// TIA Portal V17 program export: 2 tag tables, 3 data types, 1 data blocks, 4 code blocks (in call order from the OBs), 2 instance data blocks

VAR_GLOBAL   // PLC tag table "Default tag table"
END_VAR

VAR_GLOBAL   // PLC tag table "LPMLV2022_Constants"
END_VAR
VAR_GLOBAL CONSTANT   // user constants
   LPMLV2022_MODE_INVALID : DInt := 0;   // OMAC PackMLV2022 unit mode Invalid
   LPMLV2022_MODE_PRODUCTION : DInt := 1;   // OMAC PackMLV2022 unit mode Production
   LPMLV2022_MODE_MAINTENANCE : DInt := 2;   // OMAC PackMLV2022 unit mode Maintenance
   LPMLV2022_MODE_MANUAL : DInt := 3;   // OMAC PackMLV2022 unit mode Manual
   LPMLV2022_MODE_USER_01 : DInt := 4;   // OMAC PackMLV2022 user-defined unit mode 01
   LPMLV2022_MODE_USER_02 : DInt := 5;   // OMAC PackMLV2022 user-defined unit mode 02
   LPMLV2022_MODE_USER_03 : DInt := 6;   // OMAC PackMLV2022 user-defined unit mode 03
   LPMLV2022_MODE_USER_04 : DInt := 7;   // OMAC PackMLV2022 user-defined unit mode 04
   LPMLV2022_MODE_USER_05 : DInt := 8;   // OMAC PackMLV2022 user-defined unit mode 05
   LPMLV2022_MODE_USER_06 : DInt := 9;   // OMAC PackMLV2022 user-defined unit mode 06
   LPMLV2022_MODE_USER_07 : DInt := 10;   // OMAC PackMLV2022 user-defined unit mode 07
   LPMLV2022_MODE_USER_08 : DInt := 11;   // OMAC PackMLV2022 user-defined unit mode 08
   LPMLV2022_MODE_USER_09 : DInt := 12;   // OMAC PackMLV2022 user-defined unit mode 09
   LPMLV2022_MODE_USER_10 : DInt := 13;   // OMAC PackMLV2022 user-defined unit mode 10
   LPMLV2022_MODE_USER_11 : DInt := 14;   // OMAC PackMLV2022 user-defined unit mode 11
   LPMLV2022_MODE_USER_12 : DInt := 15;   // OMAC PackMLV2022 user-defined unit mode 12
   LPMLV2022_MODE_USER_13 : DInt := 16;   // OMAC PackMLV2022 user-defined unit mode 13
   LPMLV2022_MODE_USER_14 : DInt := 17;   // OMAC PackMLV2022 user-defined unit mode 14
   LPMLV2022_MODE_USER_15 : DInt := 18;   // OMAC PackMLV2022 user-defined unit mode 15
   LPMLV2022_MODE_USER_16 : DInt := 19;   // OMAC PackMLV2022 user-defined unit mode 16
   LPMLV2022_MODE_USER_17 : DInt := 20;   // OMAC PackMLV2022 user-defined unit mode 17
   LPMLV2022_MODE_USER_18 : DInt := 21;   // OMAC PackMLV2022 user-defined unit mode 18
   LPMLV2022_MODE_USER_19 : DInt := 22;   // OMAC PackMLV2022 user-defined unit mode 19
   LPMLV2022_MODE_USER_20 : DInt := 23;   // OMAC PackMLV2022 user-defined unit mode 20
   LPMLV2022_MODE_USER_21 : DInt := 24;   // OMAC PackMLV2022 user-defined unit mode 21
   LPMLV2022_MODE_USER_22 : DInt := 25;   // OMAC PackMLV2022 user-defined unit mode 22
   LPMLV2022_MODE_USER_23 : DInt := 26;   // OMAC PackMLV2022 user-defined unit mode 23
   LPMLV2022_MODE_USER_24 : DInt := 27;   // OMAC PackMLV2022 user-defined unit mode 24
   LPMLV2022_MODE_USER_25 : DInt := 28;   // OMAC PackMLV2022 user-defined unit mode 25
   LPMLV2022_MODE_USER_26 : DInt := 29;   // OMAC PackMLV2022 user-defined unit mode 26
   LPMLV2022_MODE_USER_27 : DInt := 30;   // OMAC PackMLV2022 user-defined unit mode 27
   LPMLV2022_MODE_USER_28 : DInt := 31;   // OMAC PackMLV2022 user-defined unit mode 28
   LPMLV2022_STATE_UNDEFINED : DInt := 0;   // OMAC PackMLV2022 state Undefined
   LPMLV2022_STATE_CLEARING : DInt := 1;   // OMAC PackMLV2022 state Clearing
   LPMLV2022_STATE_STOPPED : DInt := 2;   // OMAC PackMLV2022 state Stopped
   LPMLV2022_STATE_STARTING : DInt := 3;   // OMAC PackMLV2022 state Starting
   LPMLV2022_STATE_IDLE : DInt := 4;   // OMAC PackMLV2022 state Idle
   LPMLV2022_STATE_SUSPENDED : DInt := 5;   // OMAC PackMLV2022 state Suspended
   LPMLV2022_STATE_EXECUTE : DInt := 6;   // OMAC PackMLV2022 state Execute
   LPMLV2022_STATE_STOPPING : DInt := 7;   // OMAC PackMLV2022 state Stopping
   LPMLV2022_STATE_ABORTING : DInt := 8;   // OMAC PackMLV2022 state Aborting
   LPMLV2022_STATE_ABORTED : DInt := 9;   // OMAC PackMLV2022 state Aborted
   LPMLV2022_STATE_HOLDING : DInt := 10;   // OMAC PackMLV2022 state Holding
   LPMLV2022_STATE_HELD : DInt := 11;   // OMAC PackMLV2022 state Held
   LPMLV2022_STATE_UNHOLDING : DInt := 12;   // OMAC PackMLV2022 state Unholding
   LPMLV2022_STATE_SUSPENDING : DInt := 13;   // OMAC PackMLV2022 state Suspending
   LPMLV2022_STATE_UNSUSPENDING : DInt := 14;   // OMAC PackMLV2022 state Unsuspending
   LPMLV2022_STATE_RESETTING : DInt := 15;   // OMAC PackMLV2022 state Resetting
   LPMLV2022_STATE_COMPLETING : DInt := 16;   // OMAC PackMLV2022 state Completing
   LPMLV2022_STATE_COMPLETED : DInt := 17;   // OMAC PackMLV2022 state Completed
   LPMLV2022_CMD_UNDEFINED : DInt := 0;   // OMAC PackMLV2022 control command Undefined
   LPMLV2022_CMD_RESET : DInt := 1;   // OMAC PackMLV2022 control command Reset
   LPMLV2022_CMD_START : DInt := 2;   // OMAC PackMLV2022 control command Start
   LPMLV2022_CMD_STOP : DInt := 3;   // OMAC PackMLV2022 control command Stop
   LPMLV2022_CMD_HOLD : DInt := 4;   // OMAC PackMLV2022 control command Hold
   LPMLV2022_CMD_UNHOLD : DInt := 5;   // OMAC PackMLV2022 control command Unhold
   LPMLV2022_CMD_SUSPEND : DInt := 6;   // OMAC PackMLV2022 control command Suspend
   LPMLV2022_CMD_UNSUSPEND : DInt := 7;   // OMAC PackMLV2022 control command Unsuspend
   LPMLV2022_CMD_ABORT : DInt := 8;   // OMAC PackMLV2022 control command Abort
   LPMLV2022_CMD_CLEAR : DInt := 9;   // OMAC PackMLV2022 control command Clear
   LPMLV2022_CMD_COMPLETE : DInt := 10;   // OMAC PackMLV2022 control command Complete
   LPMLV2022_DIAG_BUFFER_UPPER_LIM : Int := 7;   // Diagnostics buffer array upper boundary (0-based)
   LPMLV2022_MODES_UPPER_LIM : Int := 8;   // (Number of unit modes - 1) -> Array[0..LPMLV2022_MODES_UPPER_LIM]
   LPMLV2022_STATES_UPPER_LIM : Int := 17;   // (Number of states - 1) -> Array[0..LPMLV2022_STATES_UPPER_LIM]
   LPMLV2022_MAX_MODES_UPPER_LIM : Int := 31;   // (Maximum number of unit modes - 1) -> Array[0..LPMLV2022_MAX_MODES_UPPER_LIM]
END_VAR

TYPE "LPMLV2022_typeConfiguration"
TITLE = LPMLV2022_typeConfiguration
// Support: tech.team.motioncontrol@siemens.com
// stored: IsFailsafeCompliant false
   STRUCT
      EnabledModesCfg : DWord := 16#0000_01FE;   // Bit locations within the DWORD represent Mode numbers. A value of 1 in a bit location [0-31] indicates that the corresponding Mode number is enabled. Mode 0 is an Invalid Mode, therefore bit 0 is unused
      DisabledStatesCfg : Array[0.."LPMLV2022_MAX_MODES_UPPER_LIM"] of DWord;   // The array index represents the Mode number. Bit locations within the DWORD value represent State numbers. A value of 1 in a bit location indicates that the corresponding state number is disabled. State 0 is an Undefined State, therefore bit 0 is unused
      ModeTransitionCfg : Array[0.."LPMLV2022_MAX_MODES_UPPER_LIM"] of DWord;   // The array index represents the Mode number. Bit locations within the DWORD value represent State numbers. A value of 1 in a bit location indicates that a mode transition from the corresponding state number is allowed
      holdCmdCfg : DWord := 16#0000_0060;   // Bit locations within the DWORD value represent State numbers. A value of 1 in a bit location indicates that the Hold control command is taken into account in the corresponding state. Note: a state change is only performed if the Holding/Held states are not disabled. The 'holdCmdCfg' can only be activated for the following states: Idle, Starting, Execute, Completing, Completed, Suspending, Suspended, Unsuspending, Unholding
      completeCmdCfg : DWord := 16#0000_0860;   // Bit locations within the DWORD value represent State numbers. A value of 1 in a bit location indicates that the Complete control command is taken into account in the corresponding state. Note: a state change is only performed if the Completing/Completed states are not disabled. The 'completeCmdCfg' can only be activated for the following states: Execute, Suspended, Held
   END_STRUCT;
   // ModeTransitionCfg[1..31] := 16#0000_0214;
END_TYPE

TYPE "LPMLV2022_typeDiagnostics"
TITLE = LPMLV2022_typeDiagnostics
// Support: tech.team.motioncontrol@siemens.com
// stored: IsFailsafeCompliant false
   STRUCT
      bufferIndex { ExternalWritable := 'False'} : Int := -1;   // Index of actual buffer entry
      buffer { ExternalWritable := 'False'} : Array[0.."LPMLV2022_DIAG_BUFFER_UPPER_LIM"] of "LPMLV2022_typeDiagnosticsEntry";   // Diagnostics information buffer
   END_STRUCT;
END_TYPE

TYPE "LPMLV2022_typeDiagnosticsEntry"
TITLE = LPMLV2022_typeDiagnosticsEntry
// Support: tech.team.motioncontrol@siemens.com
// stored: IsFailsafeCompliant false
   STRUCT
      timestamp { ExternalWritable := 'False'} : DTL;   // Timestamp for this entry
      UnitModeCurrent { ExternalWritable := 'False'} : SInt;   // Current unit mode
      StateCurrent { ExternalWritable := 'False'} : SInt;   // Current state
      UnitMode { ExternalWritable := 'False'} : SInt;   // Requested unit mode
      CntrlCmd { ExternalWritable := 'False'} : SInt;   // Request control command
      SC { ExternalWritable := 'False'} : Bool;   // State complete signal
      message { ExternalWritable := 'False'} : Byte;   // Message for this entry
   END_STRUCT;
END_TYPE

DATA_BLOCK "GlobalData"   // DB30136
TITLE = GlobalData
{ S7_Optimized_Access := 'TRUE' }
VERSION : 0.1
// stored: AutoNumber true, DBAccessibleFromOPCUA true, IsOnlyStoredInLoadMemory false, IsRetainMemResEnabled false, IsWriteProtectedInAS false, MemoryReserve 0
   VAR
      ProductionModeRequest : Bool;   // Rising edge: Request change to unit mode Production
      MaintenanceModeRequest : Bool;   // Rising edge: Request change to unit mode Maintenance
      ManualModeRequest : Bool;   // Rising edge: Request change to unit mode Manual
      UserMode01Request : Bool;   // Rising edge: Request change to user-defined unit mode 01
      UserMode02Request : Bool;   // Rising edge: Request change to user-defined unit mode 02
      UserMode03Request : Bool;   // Rising edge: Request change to user-defined unit mode 03
      UserMode04Request : Bool;   // Rising edge: Request change to user-defined unit mode 04
      UserMode05Request : Bool;   // Rising edge: Request change to user-defined unit mode 05
      ResetCmdRequest : Bool;   // Rising edge: Request control command Reset
      StartCmdRequest : Bool;   // Rising edge: Request control command Start
      StopCmdRequest : Bool;   // Rising edge: Request control command Stop
      HoldCmdRequest : Bool;   // Rising edge: Request control command Hold
      UnholdCmdRequest : Bool;   // Rising edge: Request control command Unhold
      SuspendCmdRequest : Bool;   // Rising edge: Request control command Suspend
      UnsuspendCmdRequest : Bool;   // Rising edge: Request control command Unsuspend
      AbortCmdRequest : Bool;   // Rising edge: Request control command Abort
      ClearCmdRequest : Bool;   // Rising edge: Request control command Clear
      CompleteCmdRequest : Bool;   // Rising edge: Request control command Complete
   END_VAR
BEGIN
END_DATA_BLOCK

ORGANIZATION_BLOCK "Main"   // OB1, LAD, ProgramCycle
TITLE = "Main Program Sweep (Cycle)"
{ S7_Optimized_Access := 'TRUE' }
VERSION : 0.1
// stored: AutoNumber true, IsIECCheckEnabled false, SetENOAutomatically false
   VAR_INPUT
      Initial_Call : Bool;   // Initial call of this OB
      Remanence : Bool;   // =True, if remanent data are available
   END_VAR
BEGIN

REGION Network 1: Example of calling LPMLV2022_UnitModeStateManagerBool incl. ToDo structure
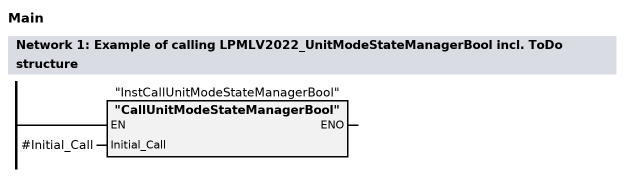
   RUNG wire#powerrail
      "InstCallUnitModeStateManagerBool"(Initial_Call := #Initial_Call)
   END_RUNG
   // the same network as SCL:
   "InstCallUnitModeStateManagerBool"(Initial_Call := #Initial_Call);   // "CallUnitModeStateManagerBool"
END_REGION
END_ORGANIZATION_BLOCK

FUNCTION_BLOCK "CallUnitModeStateManagerBool"   // FB30133, LAD
{ S7_Optimized_Access := 'TRUE' }
VERSION : 0.1
// stored: AutoNumber true, IsIECCheckEnabled false, IsRetainMemResEnabled false, MemoryReserve 0, SetENOAutomatically false, UDAEnableTagReadback false
   VAR_INPUT
      Initial_Call { ExternalAccessible := 'False'; ExternalVisible := 'False'; ExternalWritable := 'False'} : Bool;   // Initial call flag from the calling OB
   END_VAR
   VAR_TEMP
      tempUnitModeCurrent : UInt;   // Current unit mode for jump list
      tempStateCurrent : UInt;   // Current state for jump list
      tempDummy : Bool;   // Dummy
   END_VAR
BEGIN

REGION Network 1: First cycle: Disable unit modes and set state configuration in modes - default: Base state model
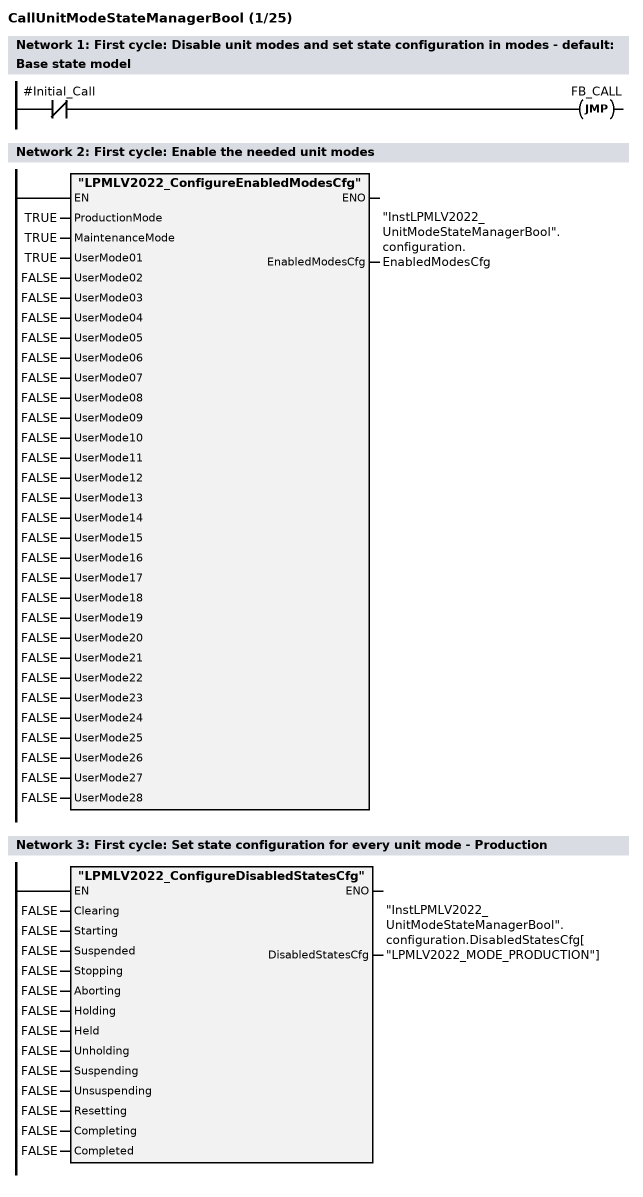
   RUNG wire#powerrail
      I_Contact( #Initial_Call )
      JumpCoil( FB_CALL )
   END_RUNG
   // the same network as SCL:
   IF NOT #Initial_Call THEN GOTO FB_CALL; END_IF;
END_REGION

REGION Network 2: First cycle: Enable the needed unit modes
   RUNG wire#powerrail
      "LPMLV2022_ConfigureEnabledModesCfg"(ProductionMode := TRUE, MaintenanceMode := TRUE, UserMode01 := TRUE, UserMode02 := FALSE, UserMode03 := FALSE, UserMode04 := FALSE, UserMode05 := FALSE, UserMode06 := FALSE, UserMode07 := FALSE, UserMode08 := FALSE, UserMode09 := FALSE, UserMode10 := FALSE, UserMode11 := FALSE, UserMode12 := FALSE, UserMode13 := FALSE, UserMode14 := FALSE, UserMode15 := FALSE, UserMode16 := FALSE, UserMode17 := FALSE, UserMode18 := FALSE, UserMode19 := FALSE, UserMode20 := FALSE, UserMode21 := FALSE, UserMode22 := FALSE, UserMode23 := FALSE, UserMode24 := FALSE, UserMode25 := FALSE, UserMode26 := FALSE, UserMode27 := FALSE, UserMode28 := FALSE, EnabledModesCfg => "InstLPMLV2022_UnitModeStateManagerBool".configuration.EnabledModesCfg)
   END_RUNG
   // the same network as SCL:
   "LPMLV2022_ConfigureEnabledModesCfg"(ProductionMode := TRUE,
                           MaintenanceMode := TRUE,
                           UserMode01 := TRUE,
                           UserMode02 := FALSE,
                           UserMode03 := FALSE,
                           UserMode04 := FALSE,
                           UserMode05 := FALSE,
                           UserMode06 := FALSE,
                           UserMode07 := FALSE,
                           UserMode08 := FALSE,
                           UserMode09 := FALSE,
                           UserMode10 := FALSE,
                           UserMode11 := FALSE,
                           UserMode12 := FALSE,
                           UserMode13 := FALSE,
                           UserMode14 := FALSE,
                           UserMode15 := FALSE,
                           UserMode16 := FALSE,
                           UserMode17 := FALSE,
                           UserMode18 := FALSE,
                           UserMode19 := FALSE,
                           UserMode20 := FALSE,
                           UserMode21 := FALSE,
                           UserMode22 := FALSE,
                           UserMode23 := FALSE,
                           UserMode24 := FALSE,
                           UserMode25 := FALSE,
                           UserMode26 := FALSE,
                           UserMode27 := FALSE,
                           UserMode28 := FALSE,
                           EnabledModesCfg => "InstLPMLV2022_UnitModeStateManagerBool".configuration.EnabledModesCfg);
END_REGION

REGION Network 3: First cycle: Set state configuration for every unit mode - Production
   RUNG wire#powerrail
      "LPMLV2022_ConfigureDisabledStatesCfg"(Clearing := FALSE, Starting := FALSE, Suspended := FALSE, Stopping := FALSE, Aborting := FALSE, Holding := FALSE, Held := FALSE, Unholding := FALSE, Suspending := FALSE, Unsuspending := FALSE, Resetting := FALSE, Completing := FALSE, Completed := FALSE, DisabledStatesCfg => "InstLPMLV2022_UnitModeStateManagerBool".configuration.DisabledStatesCfg["LPMLV2022_MODE_PRODUCTION"])
   END_RUNG
   // the same network as SCL:
   "LPMLV2022_ConfigureDisabledStatesCfg"(Clearing := FALSE,
                           Starting := FALSE,
                           Suspended := FALSE,
                           Stopping := FALSE,
                           Aborting := FALSE,
                           Holding := FALSE,
                           Held := FALSE,
                           Unholding := FALSE,
                           Suspending := FALSE,
                           Unsuspending := FALSE,
                           Resetting := FALSE,
                           Completing := FALSE,
                           Completed := FALSE,
                           DisabledStatesCfg => "InstLPMLV2022_UnitModeStateManagerBool".configuration.DisabledStatesCfg["LPMLV2022_MODE_PRODUCTION"]);
END_REGION

REGION Network 4: First cycle: Set state configuration for every unit mode - Maintenance
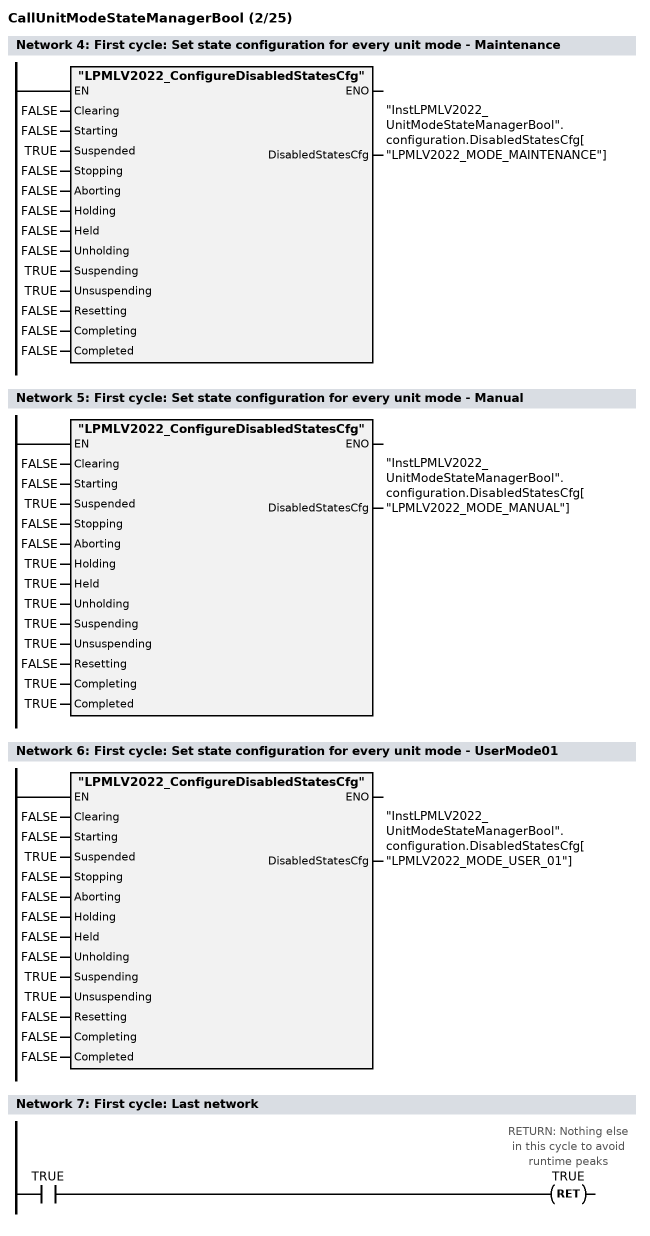
   RUNG wire#powerrail
      "LPMLV2022_ConfigureDisabledStatesCfg"(Clearing := FALSE, Starting := FALSE, Suspended := TRUE, Stopping := FALSE, Aborting := FALSE, Holding := FALSE, Held := FALSE, Unholding := FALSE, Suspending := TRUE, Unsuspending := TRUE, Resetting := FALSE, Completing := FALSE, Completed := FALSE, DisabledStatesCfg => "InstLPMLV2022_UnitModeStateManagerBool".configuration.DisabledStatesCfg["LPMLV2022_MODE_MAINTENANCE"])
   END_RUNG
   // the same network as SCL:
   "LPMLV2022_ConfigureDisabledStatesCfg"(Clearing := FALSE,
                           Starting := FALSE,
                           Suspended := TRUE,
                           Stopping := FALSE,
                           Aborting := FALSE,
                           Holding := FALSE,
                           Held := FALSE,
                           Unholding := FALSE,
                           Suspending := TRUE,
                           Unsuspending := TRUE,
                           Resetting := FALSE,
                           Completing := FALSE,
                           Completed := FALSE,
                           DisabledStatesCfg => "InstLPMLV2022_UnitModeStateManagerBool".configuration.DisabledStatesCfg["LPMLV2022_MODE_MAINTENANCE"]);
END_REGION

REGION Network 5: First cycle: Set state configuration for every unit mode - Manual
   RUNG wire#powerrail
      "LPMLV2022_ConfigureDisabledStatesCfg"(Clearing := FALSE, Starting := FALSE, Suspended := TRUE, Stopping := FALSE, Aborting := FALSE, Holding := TRUE, Held := TRUE, Unholding := TRUE, Suspending := TRUE, Unsuspending := TRUE, Resetting := FALSE, Completing := TRUE, Completed := TRUE, DisabledStatesCfg => "InstLPMLV2022_UnitModeStateManagerBool".configuration.DisabledStatesCfg["LPMLV2022_MODE_MANUAL"])
   END_RUNG
   // the same network as SCL:
   "LPMLV2022_ConfigureDisabledStatesCfg"(Clearing := FALSE,
                           Starting := FALSE,
                           Suspended := TRUE,
                           Stopping := FALSE,
                           Aborting := FALSE,
                           Holding := TRUE,
                           Held := TRUE,
                           Unholding := TRUE,
                           Suspending := TRUE,
                           Unsuspending := TRUE,
                           Resetting := FALSE,
                           Completing := TRUE,
                           Completed := TRUE,
                           DisabledStatesCfg => "InstLPMLV2022_UnitModeStateManagerBool".configuration.DisabledStatesCfg["LPMLV2022_MODE_MANUAL"]);
END_REGION

REGION Network 6: First cycle: Set state configuration for every unit mode - UserMode01
   RUNG wire#powerrail
      "LPMLV2022_ConfigureDisabledStatesCfg"(Clearing := FALSE, Starting := FALSE, Suspended := TRUE, Stopping := FALSE, Aborting := FALSE, Holding := FALSE, Held := FALSE, Unholding := FALSE, Suspending := TRUE, Unsuspending := TRUE, Resetting := FALSE, Completing := FALSE, Completed := FALSE, DisabledStatesCfg => "InstLPMLV2022_UnitModeStateManagerBool".configuration.DisabledStatesCfg["LPMLV2022_MODE_USER_01"])
   END_RUNG
   // the same network as SCL:
   "LPMLV2022_ConfigureDisabledStatesCfg"(Clearing := FALSE,
                           Starting := FALSE,
                           Suspended := TRUE,
                           Stopping := FALSE,
                           Aborting := FALSE,
                           Holding := FALSE,
                           Held := FALSE,
                           Unholding := FALSE,
                           Suspending := TRUE,
                           Unsuspending := TRUE,
                           Resetting := FALSE,
                           Completing := FALSE,
                           Completed := FALSE,
                           DisabledStatesCfg => "InstLPMLV2022_UnitModeStateManagerBool".configuration.DisabledStatesCfg["LPMLV2022_MODE_USER_01"]);
END_REGION

REGION Network 7: First cycle: Last network
   RUNG wire#powerrail
      Contact( TRUE )
      ReturnCoil( TRUE )
   END_RUNG
   // the same network as SCL:
   IF TRUE THEN
       ENO := TRUE;   // RETURN: Nothing else in this cycle to avoid runtime peaks
       RETURN;
   END_IF;
END_REGION

REGION Network 8: Call of LPMLV2022_UnitModeStateManagerBool
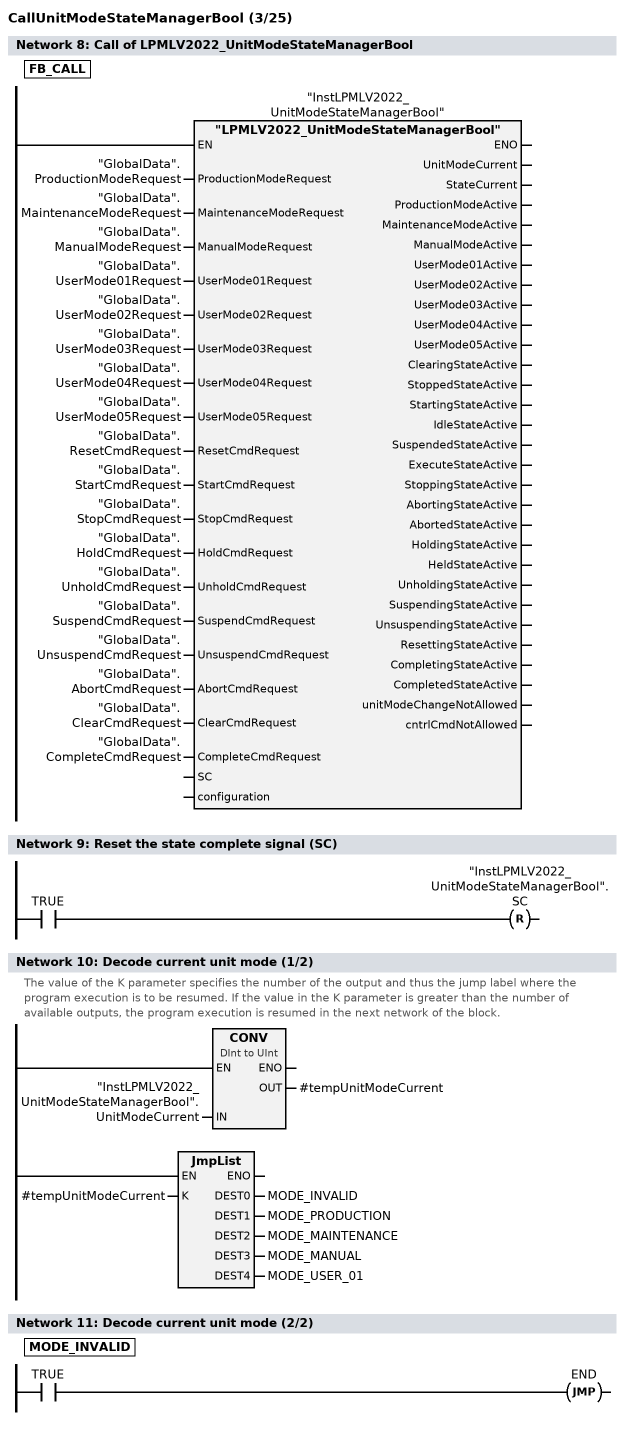
   Label( FB_CALL )
   RUNG wire#powerrail
      "InstLPMLV2022_UnitModeStateManagerBool"(ProductionModeRequest := "GlobalData".ProductionModeRequest, MaintenanceModeRequest := "GlobalData".MaintenanceModeRequest, ManualModeRequest := "GlobalData".ManualModeRequest, UserMode01Request := "GlobalData".UserMode01Request, UserMode02Request := "GlobalData".UserMode02Request, UserMode03Request := "GlobalData".UserMode03Request, UserMode04Request := "GlobalData".UserMode04Request, UserMode05Request := "GlobalData".UserMode05Request, ResetCmdRequest := "GlobalData".ResetCmdRequest, StartCmdRequest := "GlobalData".StartCmdRequest, StopCmdRequest := "GlobalData".StopCmdRequest, HoldCmdRequest := "GlobalData".HoldCmdRequest, UnholdCmdRequest := "GlobalData".UnholdCmdRequest, SuspendCmdRequest := "GlobalData".SuspendCmdRequest, UnsuspendCmdRequest := "GlobalData".UnsuspendCmdRequest, AbortCmdRequest := "GlobalData".AbortCmdRequest, ClearCmdRequest := "GlobalData".ClearCmdRequest, CompleteCmdRequest := "GlobalData".CompleteCmdRequest, SC :=, configuration :=, UnitModeCurrent =>, StateCurrent =>, ProductionModeActive =>, MaintenanceModeActive =>, ManualModeActive =>, UserMode01Active =>, UserMode02Active =>, UserMode03Active =>, UserMode04Active =>, UserMode05Active =>, ClearingStateActive =>, StoppedStateActive =>, StartingStateActive =>, IdleStateActive =>, SuspendedStateActive =>, ExecuteStateActive =>, StoppingStateActive =>, AbortingStateActive =>, AbortedStateActive =>, HoldingStateActive =>, HeldStateActive =>, UnholdingStateActive =>, SuspendingStateActive =>, UnsuspendingStateActive =>, ResettingStateActive =>, CompletingStateActive =>, CompletedStateActive =>, unitModeChangeNotAllowed =>, cntrlCmdNotAllowed =>)
   END_RUNG
   // the same network as SCL:
   FB_CALL:
   "InstLPMLV2022_UnitModeStateManagerBool"(ProductionModeRequest := "GlobalData".ProductionModeRequest,   // "LPMLV2022_UnitModeStateManagerBool"
                           MaintenanceModeRequest := "GlobalData".MaintenanceModeRequest,
                           ManualModeRequest := "GlobalData".ManualModeRequest,
                           UserMode01Request := "GlobalData".UserMode01Request,
                           UserMode02Request := "GlobalData".UserMode02Request,
                           UserMode03Request := "GlobalData".UserMode03Request,
                           UserMode04Request := "GlobalData".UserMode04Request,
                           UserMode05Request := "GlobalData".UserMode05Request,
                           ResetCmdRequest := "GlobalData".ResetCmdRequest,
                           StartCmdRequest := "GlobalData".StartCmdRequest,
                           StopCmdRequest := "GlobalData".StopCmdRequest,
                           HoldCmdRequest := "GlobalData".HoldCmdRequest,
                           UnholdCmdRequest := "GlobalData".UnholdCmdRequest,
                           SuspendCmdRequest := "GlobalData".SuspendCmdRequest,
                           UnsuspendCmdRequest := "GlobalData".UnsuspendCmdRequest,
                           AbortCmdRequest := "GlobalData".AbortCmdRequest,
                           ClearCmdRequest := "GlobalData".ClearCmdRequest,
                           CompleteCmdRequest := "GlobalData".CompleteCmdRequest);
END_REGION

REGION Network 9: Reset the state complete signal (SC)
   RUNG wire#powerrail
      Contact( TRUE )
      R_Coil( "InstLPMLV2022_UnitModeStateManagerBool".SC )
   END_RUNG
   // the same network as SCL:
   IF TRUE THEN "InstLPMLV2022_UnitModeStateManagerBool".SC := FALSE; END_IF;
END_REGION

REGION Network 10: Decode current unit mode (1/2)
   // The value of the K parameter specifies the number of the output and thus the jump label where the program execution is to be resumed. If the value in the K parameter is greater than the number of available outputs, the program execution is resumed in the next network of the block.
   // no SCL statement known for JmpList: written as a call
   #tempUnitModeCurrent := DINT_TO_UINT("InstLPMLV2022_UnitModeStateManagerBool".UnitModeCurrent);
   JmpList(k := #tempUnitModeCurrent,
           dest0 => MODE_INVALID,
           dest1 => MODE_PRODUCTION,
           dest2 => MODE_MAINTENANCE,
           dest3 => MODE_MANUAL,
           dest4 => MODE_USER_01);
END_REGION

REGION Network 11: Decode current unit mode (2/2)
   Label( MODE_INVALID )
   RUNG wire#powerrail
      Contact( TRUE )
      JumpCoil( END )
   END_RUNG
   // the same network as SCL:
   MODE_INVALID:
   IF TRUE THEN GOTO END; END_IF;
END_REGION

REGION Network 12: Unit mode Production - Decode current state for unit mode (1/2)
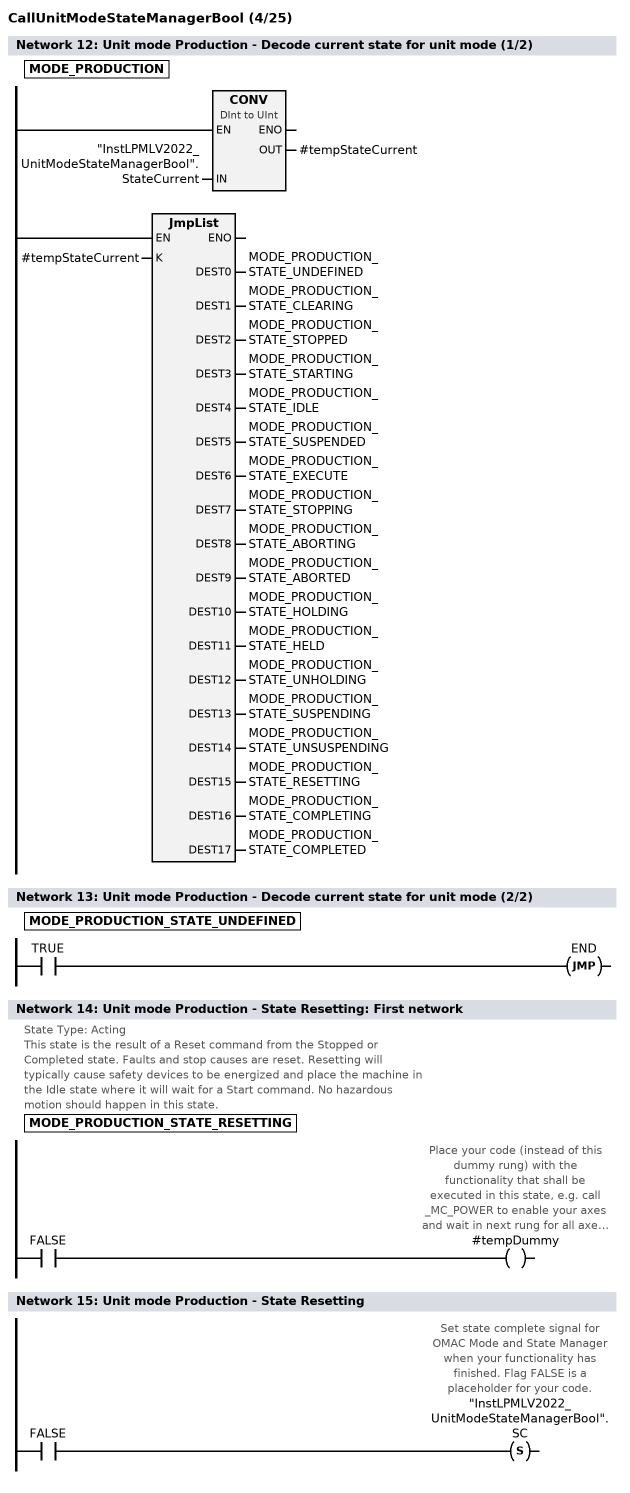
   // no SCL statement known for JmpList: written as a call
   MODE_PRODUCTION:
   #tempStateCurrent := DINT_TO_UINT("InstLPMLV2022_UnitModeStateManagerBool".StateCurrent);
   JmpList(k := #tempStateCurrent,
           dest0 => MODE_PRODUCTION_STATE_UNDEFINED,
           dest1 => MODE_PRODUCTION_STATE_CLEARING,
           dest2 => MODE_PRODUCTION_STATE_STOPPED,
           dest3 => MODE_PRODUCTION_STATE_STARTING,
           dest4 => MODE_PRODUCTION_STATE_IDLE,
           dest5 => MODE_PRODUCTION_STATE_SUSPENDED,
           dest6 => MODE_PRODUCTION_STATE_EXECUTE,
           dest7 => MODE_PRODUCTION_STATE_STOPPING,
           dest8 => MODE_PRODUCTION_STATE_ABORTING,
           dest9 => MODE_PRODUCTION_STATE_ABORTED,
           dest10 => MODE_PRODUCTION_STATE_HOLDING,
           dest11 => MODE_PRODUCTION_STATE_HELD,
           dest12 => MODE_PRODUCTION_STATE_UNHOLDING,
           dest13 => MODE_PRODUCTION_STATE_SUSPENDING,
           dest14 => MODE_PRODUCTION_STATE_UNSUSPENDING,
           dest15 => MODE_PRODUCTION_STATE_RESETTING,
           dest16 => MODE_PRODUCTION_STATE_COMPLETING,
           dest17 => MODE_PRODUCTION_STATE_COMPLETED);
END_REGION

REGION Network 13: Unit mode Production - Decode current state for unit mode (2/2)
   Label( MODE_PRODUCTION_STATE_UNDEFINED )
   RUNG wire#powerrail
      Contact( TRUE )
      JumpCoil( END )
   END_RUNG
   // the same network as SCL:
   MODE_PRODUCTION_STATE_UNDEFINED:
   IF TRUE THEN GOTO END; END_IF;
END_REGION

REGION Network 14: Unit mode Production - State Resetting: First network
   // State Type: Acting
   // This state is the result of a Reset command from the Stopped or
   // Completed state. Faults and stop causes are reset. Resetting will
   // typically cause safety devices to be energized and place the machine in
   // the Idle state where it will wait for a Start command. No hazardous
   // motion should happen in this state.
   Label( MODE_PRODUCTION_STATE_RESETTING )
   RUNG wire#powerrail
      Contact( FALSE )
      Coil( #tempDummy )   // Place your code (instead of this dummy rung) with the functionality that shall be executed in this state, e.g. call _MC_POWER to enable your axes and wait in next rung for all axes being enabled.
   END_RUNG
   // the same network as SCL:
   MODE_PRODUCTION_STATE_RESETTING:
   #tempDummy := FALSE;   // Place your code (instead of this dummy rung) with the functionality that shall be executed in this state, e.g. call _MC_POWER to enable your axes and wait in next rung for all axes being enabled.
END_REGION

REGION Network 15: Unit mode Production - State Resetting
   RUNG wire#powerrail
      Contact( FALSE )
      S_Coil( "InstLPMLV2022_UnitModeStateManagerBool".SC )   // Set state complete signal for OMAC Mode and State Manager when your functionality has finished. Flag FALSE is a placeholder for your code.
   END_RUNG
   // the same network as SCL:
   IF FALSE THEN
       "InstLPMLV2022_UnitModeStateManagerBool".SC := TRUE;   // Set state complete signal for OMAC Mode and State Manager when your functionality has finished. Flag FALSE is a placeholder for your code.
   END_IF;
END_REGION

REGION Network 16: Unit mode Production - State Resetting: Last network
   // Do not modify this network.
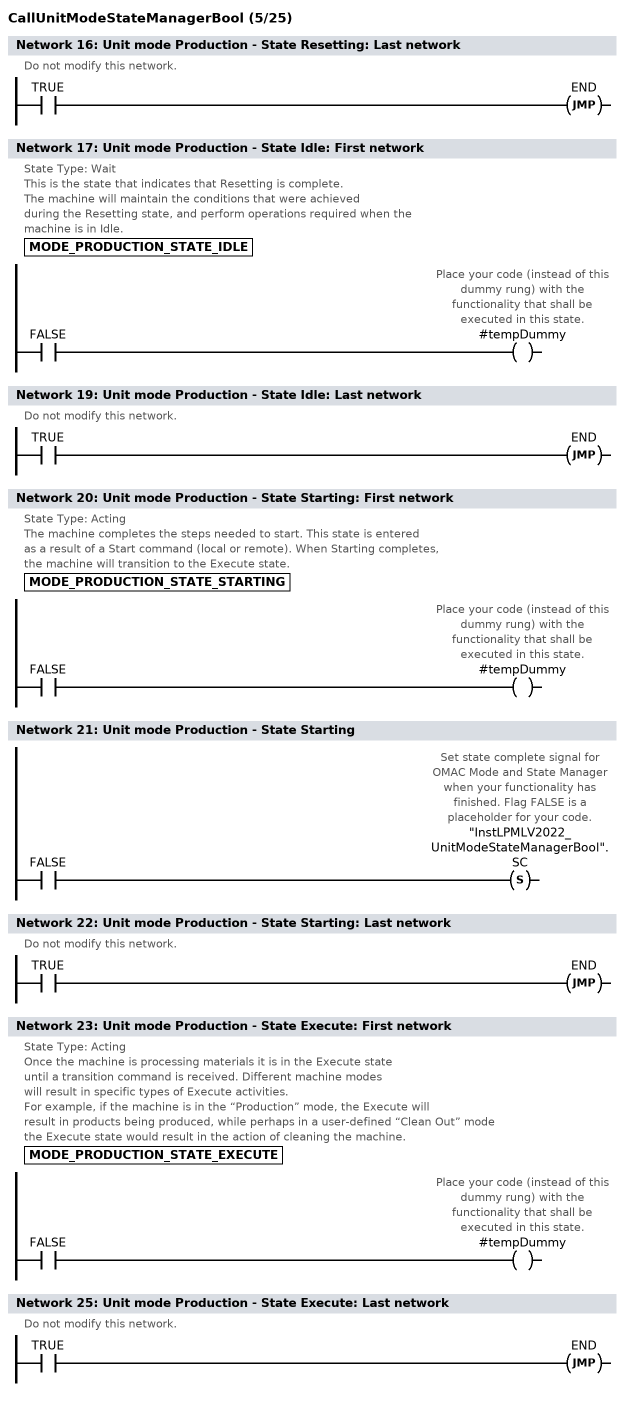
   RUNG wire#powerrail
      Contact( TRUE )
      JumpCoil( END )
   END_RUNG
   // the same network as SCL:
   IF TRUE THEN GOTO END; END_IF;
END_REGION

REGION Network 17: Unit mode Production - State Idle: First network
   // State Type: Wait
   // This is the state that indicates that Resetting is complete.
   // The machine will maintain the conditions that were achieved
   // during the Resetting state, and perform operations required when the
   // machine is in Idle.
   Label( MODE_PRODUCTION_STATE_IDLE )
   RUNG wire#powerrail
      Contact( FALSE )
      Coil( #tempDummy )   // Place your code (instead of this dummy rung) with the functionality that shall be executed in this state.
   END_RUNG
   // the same network as SCL:
   MODE_PRODUCTION_STATE_IDLE:
   #tempDummy := FALSE;   // Place your code (instead of this dummy rung) with the functionality that shall be executed in this state.
END_REGION

REGION Network 18: Unit mode Production - State Idle
END_REGION

REGION Network 19: Unit mode Production - State Idle: Last network
   // Do not modify this network.
   RUNG wire#powerrail
      Contact( TRUE )
      JumpCoil( END )
   END_RUNG
   // the same network as SCL:
   IF TRUE THEN GOTO END; END_IF;
END_REGION

REGION Network 20: Unit mode Production - State Starting: First network
   // State Type: Acting
   // The machine completes the steps needed to start. This state is entered
   // as a result of a Start command (local or remote). When Starting completes,
   // the machine will transition to the Execute state.
   Label( MODE_PRODUCTION_STATE_STARTING )
   RUNG wire#powerrail
      Contact( FALSE )
      Coil( #tempDummy )   // Place your code (instead of this dummy rung) with the functionality that shall be executed in this state.
   END_RUNG
   // the same network as SCL:
   MODE_PRODUCTION_STATE_STARTING:
   #tempDummy := FALSE;   // Place your code (instead of this dummy rung) with the functionality that shall be executed in this state.
END_REGION

REGION Network 21: Unit mode Production - State Starting
   RUNG wire#powerrail
      Contact( FALSE )
      S_Coil( "InstLPMLV2022_UnitModeStateManagerBool".SC )   // Set state complete signal for OMAC Mode and State Manager when your functionality has finished. Flag FALSE is a placeholder for your code.
   END_RUNG
   // the same network as SCL:
   IF FALSE THEN
       "InstLPMLV2022_UnitModeStateManagerBool".SC := TRUE;   // Set state complete signal for OMAC Mode and State Manager when your functionality has finished. Flag FALSE is a placeholder for your code.
   END_IF;
END_REGION

REGION Network 22: Unit mode Production - State Starting: Last network
   // Do not modify this network.
   RUNG wire#powerrail
      Contact( TRUE )
      JumpCoil( END )
   END_RUNG
   // the same network as SCL:
   IF TRUE THEN GOTO END; END_IF;
END_REGION

REGION Network 23: Unit mode Production - State Execute: First network
   // State Type: Acting
   // Once the machine is processing materials it is in the Execute state
   // until a transition command is received. Different machine modes
   // will result in specific types of Execute activities.
   // For example, if the machine is in the “Production” mode, the Execute will
   // result in products being produced, while perhaps in a user-defined “Clean Out” mode
   // the Execute state would result in the action of cleaning the machine.
   Label( MODE_PRODUCTION_STATE_EXECUTE )
   RUNG wire#powerrail
      Contact( FALSE )
      Coil( #tempDummy )   // Place your code (instead of this dummy rung) with the functionality that shall be executed in this state.
   END_RUNG
   // the same network as SCL:
   MODE_PRODUCTION_STATE_EXECUTE:
   #tempDummy := FALSE;   // Place your code (instead of this dummy rung) with the functionality that shall be executed in this state.
END_REGION

REGION Network 24: Unit mode Production - State Execute
END_REGION

REGION Network 25: Unit mode Production - State Execute: Last network
   // Do not modify this network.
   RUNG wire#powerrail
      Contact( TRUE )
      JumpCoil( END )
   END_RUNG
   // the same network as SCL:
   IF TRUE THEN GOTO END; END_IF;
END_REGION

REGION Network 26: Unit mode Production - State Stopping: First network
   // State Type: Acting
   // This state is entered in response to a Stop command.
   // While in this state the machine executes the logic that brings it to a
   // controlled stop as reflected by the Stopped state. Normal Starting
   // of the machine cannot be initiated unless Resetting has taken place.
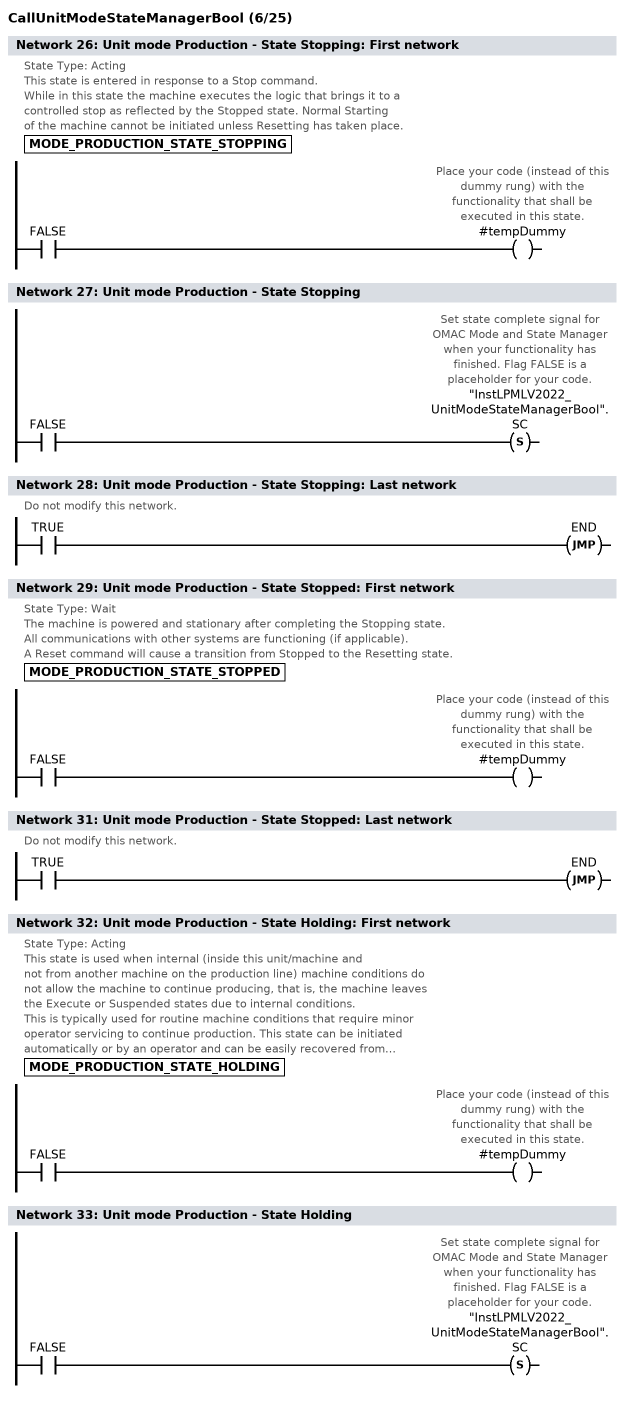
   Label( MODE_PRODUCTION_STATE_STOPPING )
   RUNG wire#powerrail
      Contact( FALSE )
      Coil( #tempDummy )   // Place your code (instead of this dummy rung) with the functionality that shall be executed in this state.
   END_RUNG
   // the same network as SCL:
   MODE_PRODUCTION_STATE_STOPPING:
   #tempDummy := FALSE;   // Place your code (instead of this dummy rung) with the functionality that shall be executed in this state.
END_REGION

REGION Network 27: Unit mode Production - State Stopping
   RUNG wire#powerrail
      Contact( FALSE )
      S_Coil( "InstLPMLV2022_UnitModeStateManagerBool".SC )   // Set state complete signal for OMAC Mode and State Manager when your functionality has finished. Flag FALSE is a placeholder for your code.
   END_RUNG
   // the same network as SCL:
   IF FALSE THEN
       "InstLPMLV2022_UnitModeStateManagerBool".SC := TRUE;   // Set state complete signal for OMAC Mode and State Manager when your functionality has finished. Flag FALSE is a placeholder for your code.
   END_IF;
END_REGION

REGION Network 28: Unit mode Production - State Stopping: Last network
   // Do not modify this network.
   RUNG wire#powerrail
      Contact( TRUE )
      JumpCoil( END )
   END_RUNG
   // the same network as SCL:
   IF TRUE THEN GOTO END; END_IF;
END_REGION

REGION Network 29: Unit mode Production - State Stopped: First network
   // State Type: Wait
   // The machine is powered and stationary after completing the Stopping state.
   // All communications with other systems are functioning (if applicable).
   // A Reset command will cause a transition from Stopped to the Resetting state.
   Label( MODE_PRODUCTION_STATE_STOPPED )
   RUNG wire#powerrail
      Contact( FALSE )
      Coil( #tempDummy )   // Place your code (instead of this dummy rung) with the functionality that shall be executed in this state.
   END_RUNG
   // the same network as SCL:
   MODE_PRODUCTION_STATE_STOPPED:
   #tempDummy := FALSE;   // Place your code (instead of this dummy rung) with the functionality that shall be executed in this state.
END_REGION

REGION Network 30: Unit mode Production - State Stopped
END_REGION

REGION Network 31: Unit mode Production - State Stopped: Last network
   // Do not modify this network.
   RUNG wire#powerrail
      Contact( TRUE )
      JumpCoil( END )
   END_RUNG
   // the same network as SCL:
   IF TRUE THEN GOTO END; END_IF;
END_REGION

REGION Network 32: Unit mode Production - State Holding: First network
   // State Type: Acting
   // This state is used when internal (inside this unit/machine and
   // not from another machine on the production line) machine conditions do
   // not allow the machine to continue producing, that is, the machine leaves
   // the Execute or Suspended states due to internal conditions.
   // This is typically used for routine machine conditions that require minor
   // operator servicing to continue production. This state can be initiated
   // automatically or by an operator and can be easily recovered from.
   // An example of this would be a machine that requires an operator to
   // periodically refill a glue dispenser or carton magazine and due to the
   // machine design, these operations cannot be performed while the machine
   // is running. Since these types of tasks are normal production operations,
   // it is not desirable to go through aborting or stopping sequences, and
   // because these functions are integral to the machine they are not
   // considered to be “external”. While in the Holding state, the machine is
   // typically brought to a controlled stop and then transitions to Held upon
   // state complete. To be able to restart production correctly after the
   // Held state, all relevant process set points and return status of the
   // procedures at the time of receiving the Hold command must be saved in
   // the machine controller when executing the Holding procedure.
   Label( MODE_PRODUCTION_STATE_HOLDING )
   RUNG wire#powerrail
      Contact( FALSE )
      Coil( #tempDummy )   // Place your code (instead of this dummy rung) with the functionality that shall be executed in this state.
   END_RUNG
   // the same network as SCL:
   MODE_PRODUCTION_STATE_HOLDING:
   #tempDummy := FALSE;   // Place your code (instead of this dummy rung) with the functionality that shall be executed in this state.
END_REGION

REGION Network 33: Unit mode Production - State Holding
   RUNG wire#powerrail
      Contact( FALSE )
      S_Coil( "InstLPMLV2022_UnitModeStateManagerBool".SC )   // Set state complete signal for OMAC Mode and State Manager when your functionality has finished. Flag FALSE is a placeholder for your code.
   END_RUNG
   // the same network as SCL:
   IF FALSE THEN
       "InstLPMLV2022_UnitModeStateManagerBool".SC := TRUE;   // Set state complete signal for OMAC Mode and State Manager when your functionality has finished. Flag FALSE is a placeholder for your code.
   END_IF;
END_REGION

REGION Network 34: Unit mode Production - State Holding: Last network
   // Do not modify this network.
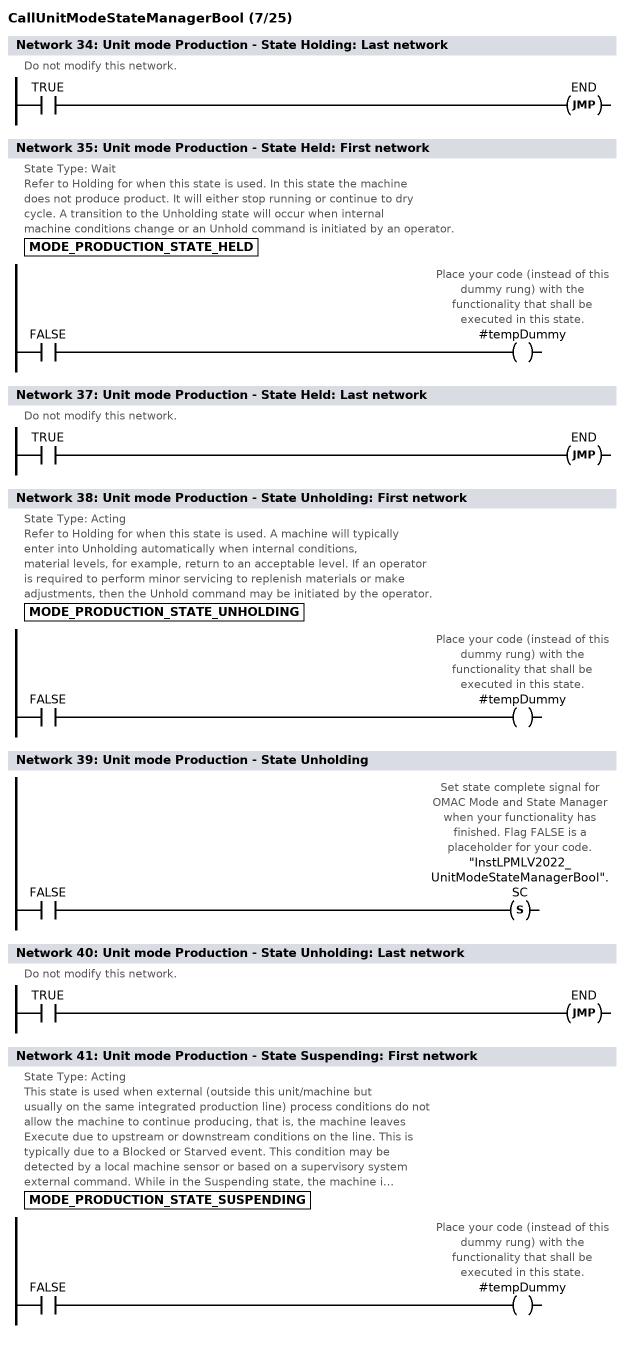
   RUNG wire#powerrail
      Contact( TRUE )
      JumpCoil( END )
   END_RUNG
   // the same network as SCL:
   IF TRUE THEN GOTO END; END_IF;
END_REGION

REGION Network 35: Unit mode Production - State Held: First network
   // State Type: Wait
   // Refer to Holding for when this state is used. In this state the machine
   // does not produce product. It will either stop running or continue to dry
   // cycle. A transition to the Unholding state will occur when internal
   // machine conditions change or an Unhold command is initiated by an operator.
   Label( MODE_PRODUCTION_STATE_HELD )
   RUNG wire#powerrail
      Contact( FALSE )
      Coil( #tempDummy )   // Place your code (instead of this dummy rung) with the functionality that shall be executed in this state.
   END_RUNG
   // the same network as SCL:
   MODE_PRODUCTION_STATE_HELD:
   #tempDummy := FALSE;   // Place your code (instead of this dummy rung) with the functionality that shall be executed in this state.
END_REGION

REGION Network 36: Unit mode Production - State Held
END_REGION

REGION Network 37: Unit mode Production - State Held: Last network
   // Do not modify this network.
   RUNG wire#powerrail
      Contact( TRUE )
      JumpCoil( END )
   END_RUNG
   // the same network as SCL:
   IF TRUE THEN GOTO END; END_IF;
END_REGION

REGION Network 38: Unit mode Production - State Unholding: First network
   // State Type: Acting
   // Refer to Holding for when this state is used. A machine will typically
   // enter into Unholding automatically when internal conditions,
   // material levels, for example, return to an acceptable level. If an operator
   // is required to perform minor servicing to replenish materials or make
   // adjustments, then the Unhold command may be initiated by the operator.
   Label( MODE_PRODUCTION_STATE_UNHOLDING )
   RUNG wire#powerrail
      Contact( FALSE )
      Coil( #tempDummy )   // Place your code (instead of this dummy rung) with the functionality that shall be executed in this state.
   END_RUNG
   // the same network as SCL:
   MODE_PRODUCTION_STATE_UNHOLDING:
   #tempDummy := FALSE;   // Place your code (instead of this dummy rung) with the functionality that shall be executed in this state.
END_REGION

REGION Network 39: Unit mode Production - State Unholding
   RUNG wire#powerrail
      Contact( FALSE )
      S_Coil( "InstLPMLV2022_UnitModeStateManagerBool".SC )   // Set state complete signal for OMAC Mode and State Manager when your functionality has finished. Flag FALSE is a placeholder for your code.
   END_RUNG
   // the same network as SCL:
   IF FALSE THEN
       "InstLPMLV2022_UnitModeStateManagerBool".SC := TRUE;   // Set state complete signal for OMAC Mode and State Manager when your functionality has finished. Flag FALSE is a placeholder for your code.
   END_IF;
END_REGION

REGION Network 40: Unit mode Production - State Unholding: Last network
   // Do not modify this network.
   RUNG wire#powerrail
      Contact( TRUE )
      JumpCoil( END )
   END_RUNG
   // the same network as SCL:
   IF TRUE THEN GOTO END; END_IF;
END_REGION

REGION Network 41: Unit mode Production - State Suspending: First network
   // State Type: Acting
   // This state is used when external (outside this unit/machine but
   // usually on the same integrated production line) process conditions do not
   // allow the machine to continue producing, that is, the machine leaves
   // Execute due to upstream or downstream conditions on the line. This is
   // typically due to a Blocked or Starved event. This condition may be
   // detected by a local machine sensor or based on a supervisory system
   // external command. While in the Suspending state, the machine is
   // typically brought to a controlled stop and then transitions to
   // Suspended upon state complete. To be able to restart production
   // correctly after the Suspended state, all relevant process set points and
   // return status of the procedures at the time of receiving the Suspend
   // command must be saved in the machine controller when executing the
   // Suspending procedure.
   Label( MODE_PRODUCTION_STATE_SUSPENDING )
   RUNG wire#powerrail
      Contact( FALSE )
      Coil( #tempDummy )   // Place your code (instead of this dummy rung) with the functionality that shall be executed in this state.
   END_RUNG
   // the same network as SCL:
   MODE_PRODUCTION_STATE_SUSPENDING:
   #tempDummy := FALSE;   // Place your code (instead of this dummy rung) with the functionality that shall be executed in this state.
END_REGION

REGION Network 42: Unit mode Production - State Suspending
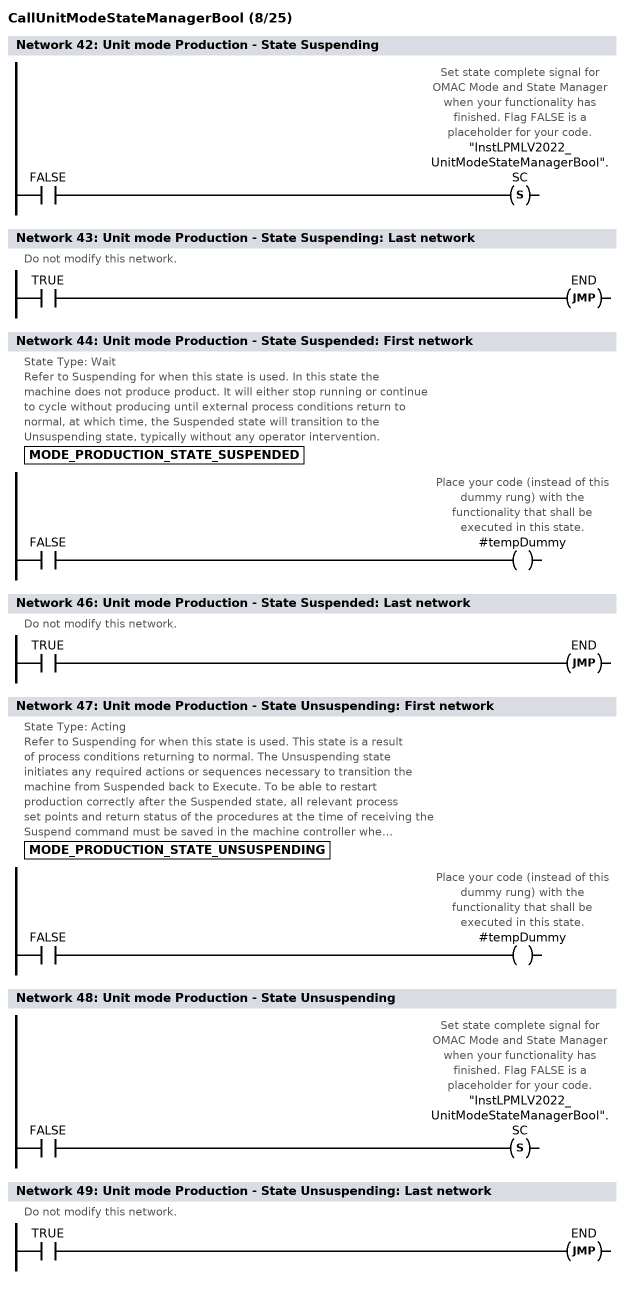
   RUNG wire#powerrail
      Contact( FALSE )
      S_Coil( "InstLPMLV2022_UnitModeStateManagerBool".SC )   // Set state complete signal for OMAC Mode and State Manager when your functionality has finished. Flag FALSE is a placeholder for your code.
   END_RUNG
   // the same network as SCL:
   IF FALSE THEN
       "InstLPMLV2022_UnitModeStateManagerBool".SC := TRUE;   // Set state complete signal for OMAC Mode and State Manager when your functionality has finished. Flag FALSE is a placeholder for your code.
   END_IF;
END_REGION

REGION Network 43: Unit mode Production - State Suspending: Last network
   // Do not modify this network.
   RUNG wire#powerrail
      Contact( TRUE )
      JumpCoil( END )
   END_RUNG
   // the same network as SCL:
   IF TRUE THEN GOTO END; END_IF;
END_REGION

REGION Network 44: Unit mode Production - State Suspended: First network
   // State Type: Wait
   // Refer to Suspending for when this state is used. In this state the
   // machine does not produce product. It will either stop running or continue
   // to cycle without producing until external process conditions return to
   // normal, at which time, the Suspended state will transition to the
   // Unsuspending state, typically without any operator intervention.
   Label( MODE_PRODUCTION_STATE_SUSPENDED )
   RUNG wire#powerrail
      Contact( FALSE )
      Coil( #tempDummy )   // Place your code (instead of this dummy rung) with the functionality that shall be executed in this state.
   END_RUNG
   // the same network as SCL:
   MODE_PRODUCTION_STATE_SUSPENDED:
   #tempDummy := FALSE;   // Place your code (instead of this dummy rung) with the functionality that shall be executed in this state.
END_REGION

REGION Network 45: Unit mode Production - State Suspended
END_REGION

REGION Network 46: Unit mode Production - State Suspended: Last network
   // Do not modify this network.
   RUNG wire#powerrail
      Contact( TRUE )
      JumpCoil( END )
   END_RUNG
   // the same network as SCL:
   IF TRUE THEN GOTO END; END_IF;
END_REGION

REGION Network 47: Unit mode Production - State Unsuspending: First network
   // State Type: Acting
   // Refer to Suspending for when this state is used. This state is a result
   // of process conditions returning to normal. The Unsuspending state
   // initiates any required actions or sequences necessary to transition the
   // machine from Suspended back to Execute. To be able to restart
   // production correctly after the Suspended state, all relevant process
   // set points and return status of the procedures at the time of receiving the
   // Suspend command must be saved in the machine controller when
   // executing the Suspending procedure.
   Label( MODE_PRODUCTION_STATE_UNSUSPENDING )
   RUNG wire#powerrail
      Contact( FALSE )
      Coil( #tempDummy )   // Place your code (instead of this dummy rung) with the functionality that shall be executed in this state.
   END_RUNG
   // the same network as SCL:
   MODE_PRODUCTION_STATE_UNSUSPENDING:
   #tempDummy := FALSE;   // Place your code (instead of this dummy rung) with the functionality that shall be executed in this state.
END_REGION

REGION Network 48: Unit mode Production - State Unsuspending
   RUNG wire#powerrail
      Contact( FALSE )
      S_Coil( "InstLPMLV2022_UnitModeStateManagerBool".SC )   // Set state complete signal for OMAC Mode and State Manager when your functionality has finished. Flag FALSE is a placeholder for your code.
   END_RUNG
   // the same network as SCL:
   IF FALSE THEN
       "InstLPMLV2022_UnitModeStateManagerBool".SC := TRUE;   // Set state complete signal for OMAC Mode and State Manager when your functionality has finished. Flag FALSE is a placeholder for your code.
   END_IF;
END_REGION

REGION Network 49: Unit mode Production - State Unsuspending: Last network
   // Do not modify this network.
   RUNG wire#powerrail
      Contact( TRUE )
      JumpCoil( END )
   END_RUNG
   // the same network as SCL:
   IF TRUE THEN GOTO END; END_IF;
END_REGION

REGION Network 50: Unit mode Production - State Completing: First network
   // State Type: Acting
   // This state is the result of a Complete command from the Execute, Held
   // or Suspended states. The Complete command may be internally generated,
   // such as reaching the end of a predefined production count where normal
   // operation has run to completion, or externally generated, such as by a
   // supervisory system. The Completing state is often used to end a 
   // production run and summarize production data.
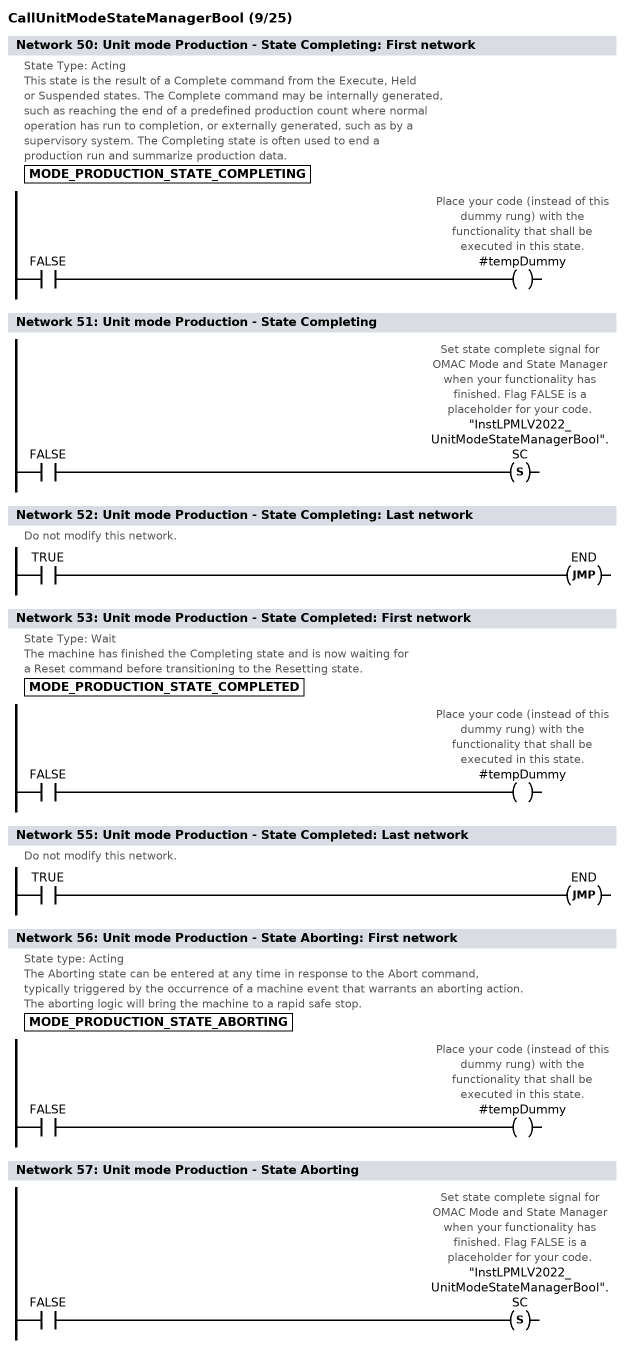
   Label( MODE_PRODUCTION_STATE_COMPLETING )
   RUNG wire#powerrail
      Contact( FALSE )
      Coil( #tempDummy )   // Place your code (instead of this dummy rung) with the functionality that shall be executed in this state.
   END_RUNG
   // the same network as SCL:
   MODE_PRODUCTION_STATE_COMPLETING:
   #tempDummy := FALSE;   // Place your code (instead of this dummy rung) with the functionality that shall be executed in this state.
END_REGION

REGION Network 51: Unit mode Production - State Completing
   RUNG wire#powerrail
      Contact( FALSE )
      S_Coil( "InstLPMLV2022_UnitModeStateManagerBool".SC )   // Set state complete signal for OMAC Mode and State Manager when your functionality has finished. Flag FALSE is a placeholder for your code.
   END_RUNG
   // the same network as SCL:
   IF FALSE THEN
       "InstLPMLV2022_UnitModeStateManagerBool".SC := TRUE;   // Set state complete signal for OMAC Mode and State Manager when your functionality has finished. Flag FALSE is a placeholder for your code.
   END_IF;
END_REGION

REGION Network 52: Unit mode Production - State Completing: Last network
   // Do not modify this network.
   RUNG wire#powerrail
      Contact( TRUE )
      JumpCoil( END )
   END_RUNG
   // the same network as SCL:
   IF TRUE THEN GOTO END; END_IF;
END_REGION

REGION Network 53: Unit mode Production - State Completed: First network
   // State Type: Wait
   // The machine has finished the Completing state and is now waiting for
   // a Reset command before transitioning to the Resetting state.
   Label( MODE_PRODUCTION_STATE_COMPLETED )
   RUNG wire#powerrail
      Contact( FALSE )
      Coil( #tempDummy )   // Place your code (instead of this dummy rung) with the functionality that shall be executed in this state.
   END_RUNG
   // the same network as SCL:
   MODE_PRODUCTION_STATE_COMPLETED:
   #tempDummy := FALSE;   // Place your code (instead of this dummy rung) with the functionality that shall be executed in this state.
END_REGION

REGION Network 54: Unit mode Production - State Completed
END_REGION

REGION Network 55: Unit mode Production - State Completed: Last network
   // Do not modify this network.
   RUNG wire#powerrail
      Contact( TRUE )
      JumpCoil( END )
   END_RUNG
   // the same network as SCL:
   IF TRUE THEN GOTO END; END_IF;
END_REGION

REGION Network 56: Unit mode Production - State Aborting: First network
   // State type: Acting
   // The Aborting state can be entered at any time in response to the Abort command,
   // typically triggered by the occurrence of a machine event that warrants an aborting action.
   // The aborting logic will bring the machine to a rapid safe stop.
   Label( MODE_PRODUCTION_STATE_ABORTING )
   RUNG wire#powerrail
      Contact( FALSE )
      Coil( #tempDummy )   // Place your code (instead of this dummy rung) with the functionality that shall be executed in this state.
   END_RUNG
   // the same network as SCL:
   MODE_PRODUCTION_STATE_ABORTING:
   #tempDummy := FALSE;   // Place your code (instead of this dummy rung) with the functionality that shall be executed in this state.
END_REGION

REGION Network 57: Unit mode Production - State Aborting
   RUNG wire#powerrail
      Contact( FALSE )
      S_Coil( "InstLPMLV2022_UnitModeStateManagerBool".SC )   // Set state complete signal for OMAC Mode and State Manager when your functionality has finished. Flag FALSE is a placeholder for your code.
   END_RUNG
   // the same network as SCL:
   IF FALSE THEN
       "InstLPMLV2022_UnitModeStateManagerBool".SC := TRUE;   // Set state complete signal for OMAC Mode and State Manager when your functionality has finished. Flag FALSE is a placeholder for your code.
   END_IF;
END_REGION

REGION Network 58: Unit mode Production - State Aborting: Last network
   // Do not modify this network.
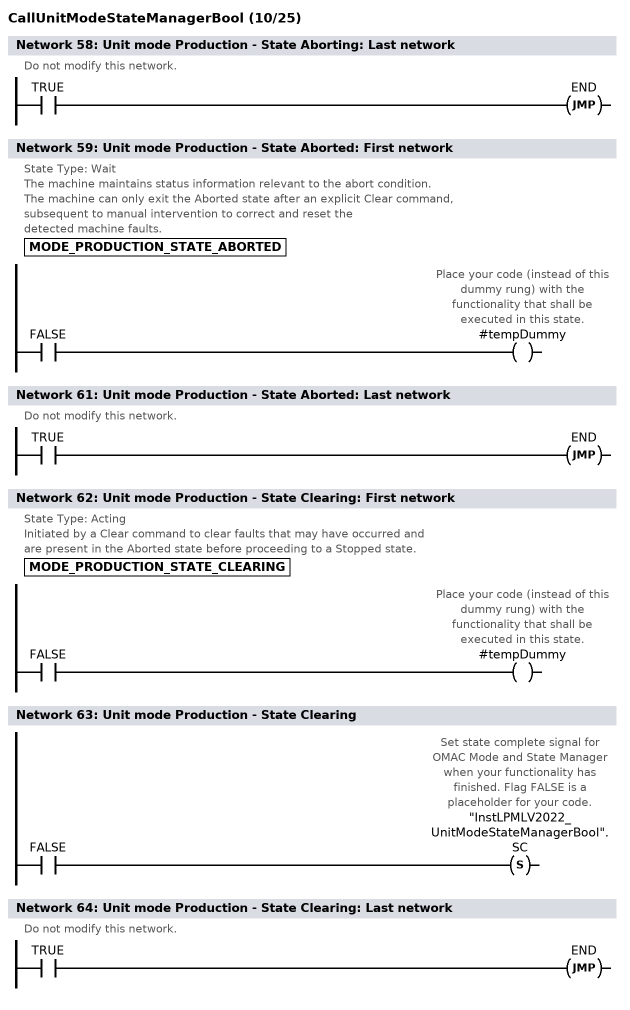
   RUNG wire#powerrail
      Contact( TRUE )
      JumpCoil( END )
   END_RUNG
   // the same network as SCL:
   IF TRUE THEN GOTO END; END_IF;
END_REGION

REGION Network 59: Unit mode Production - State Aborted: First network
   // State Type: Wait
   // The machine maintains status information relevant to the abort condition.
   // The machine can only exit the Aborted state after an explicit Clear command,
   // subsequent to manual intervention to correct and reset the
   // detected machine faults.
   Label( MODE_PRODUCTION_STATE_ABORTED )
   RUNG wire#powerrail
      Contact( FALSE )
      Coil( #tempDummy )   // Place your code (instead of this dummy rung) with the functionality that shall be executed in this state.
   END_RUNG
   // the same network as SCL:
   MODE_PRODUCTION_STATE_ABORTED:
   #tempDummy := FALSE;   // Place your code (instead of this dummy rung) with the functionality that shall be executed in this state.
END_REGION

REGION Network 60: Unit mode Production - State Aborted
END_REGION

REGION Network 61: Unit mode Production - State Aborted: Last network
   // Do not modify this network.
   RUNG wire#powerrail
      Contact( TRUE )
      JumpCoil( END )
   END_RUNG
   // the same network as SCL:
   IF TRUE THEN GOTO END; END_IF;
END_REGION

REGION Network 62: Unit mode Production - State Clearing: First network
   // State Type: Acting
   // Initiated by a Clear command to clear faults that may have occurred and
   // are present in the Aborted state before proceeding to a Stopped state.
   Label( MODE_PRODUCTION_STATE_CLEARING )
   RUNG wire#powerrail
      Contact( FALSE )
      Coil( #tempDummy )   // Place your code (instead of this dummy rung) with the functionality that shall be executed in this state.
   END_RUNG
   // the same network as SCL:
   MODE_PRODUCTION_STATE_CLEARING:
   #tempDummy := FALSE;   // Place your code (instead of this dummy rung) with the functionality that shall be executed in this state.
END_REGION

REGION Network 63: Unit mode Production - State Clearing
   RUNG wire#powerrail
      Contact( FALSE )
      S_Coil( "InstLPMLV2022_UnitModeStateManagerBool".SC )   // Set state complete signal for OMAC Mode and State Manager when your functionality has finished. Flag FALSE is a placeholder for your code.
   END_RUNG
   // the same network as SCL:
   IF FALSE THEN
       "InstLPMLV2022_UnitModeStateManagerBool".SC := TRUE;   // Set state complete signal for OMAC Mode and State Manager when your functionality has finished. Flag FALSE is a placeholder for your code.
   END_IF;
END_REGION

REGION Network 64: Unit mode Production - State Clearing: Last network
   // Do not modify this network.
   RUNG wire#powerrail
      Contact( TRUE )
      JumpCoil( END )
   END_RUNG
   // the same network as SCL:
   IF TRUE THEN GOTO END; END_IF;
END_REGION

REGION Network 65: Unit mode Maintenance - Decode current state for unit mode (1/2)
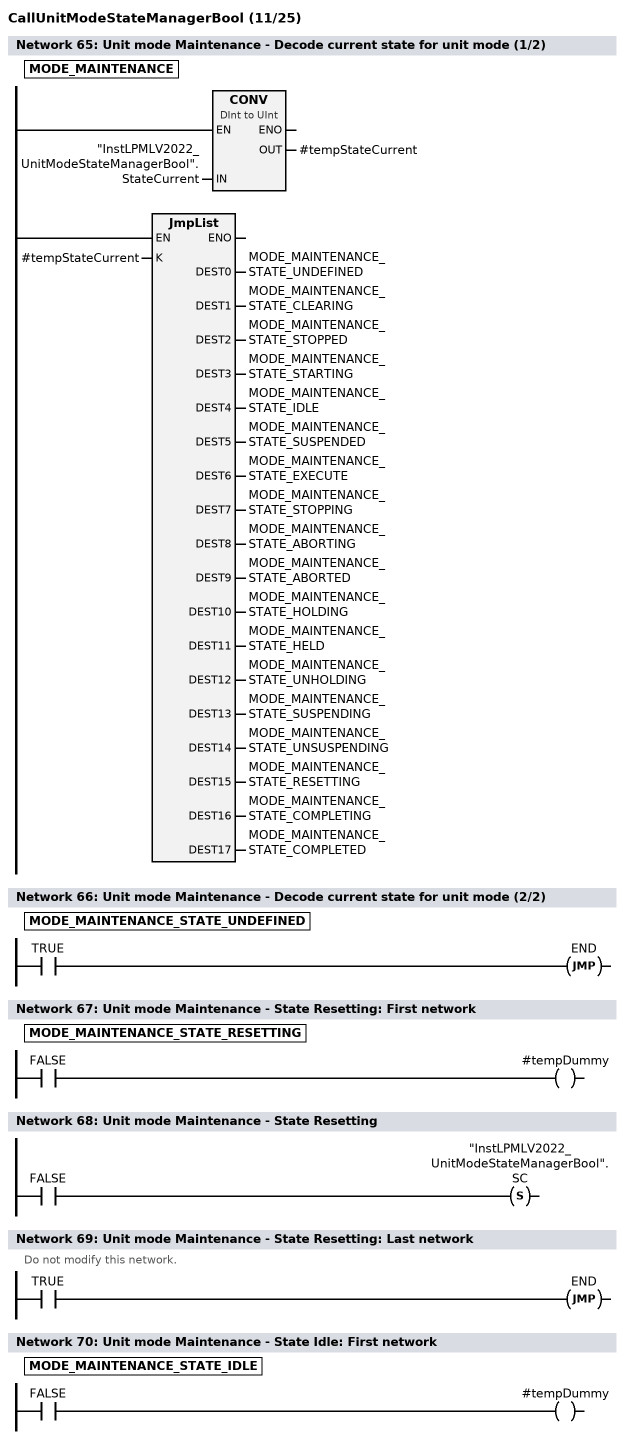
   // no SCL statement known for JmpList: written as a call
   MODE_MAINTENANCE:
   #tempStateCurrent := DINT_TO_UINT("InstLPMLV2022_UnitModeStateManagerBool".StateCurrent);
   JmpList(k := #tempStateCurrent,
           dest0 => MODE_MAINTENANCE_STATE_UNDEFINED,
           dest1 => MODE_MAINTENANCE_STATE_CLEARING,
           dest2 => MODE_MAINTENANCE_STATE_STOPPED,
           dest3 => MODE_MAINTENANCE_STATE_STARTING,
           dest4 => MODE_MAINTENANCE_STATE_IDLE,
           dest5 => MODE_MAINTENANCE_STATE_SUSPENDED,
           dest6 => MODE_MAINTENANCE_STATE_EXECUTE,
           dest7 => MODE_MAINTENANCE_STATE_STOPPING,
           dest8 => MODE_MAINTENANCE_STATE_ABORTING,
           dest9 => MODE_MAINTENANCE_STATE_ABORTED,
           dest10 => MODE_MAINTENANCE_STATE_HOLDING,
           dest11 => MODE_MAINTENANCE_STATE_HELD,
           dest12 => MODE_MAINTENANCE_STATE_UNHOLDING,
           dest13 => MODE_MAINTENANCE_STATE_SUSPENDING,
           dest14 => MODE_MAINTENANCE_STATE_UNSUSPENDING,
           dest15 => MODE_MAINTENANCE_STATE_RESETTING,
           dest16 => MODE_MAINTENANCE_STATE_COMPLETING,
           dest17 => MODE_MAINTENANCE_STATE_COMPLETED);
END_REGION

REGION Network 66: Unit mode Maintenance - Decode current state for unit mode (2/2)
   Label( MODE_MAINTENANCE_STATE_UNDEFINED )
   RUNG wire#powerrail
      Contact( TRUE )
      JumpCoil( END )
   END_RUNG
   // the same network as SCL:
   MODE_MAINTENANCE_STATE_UNDEFINED:
   IF TRUE THEN GOTO END; END_IF;
END_REGION

REGION Network 67: Unit mode Maintenance - State Resetting: First network
   Label( MODE_MAINTENANCE_STATE_RESETTING )
   RUNG wire#powerrail
      Contact( FALSE )
      Coil( #tempDummy )
   END_RUNG
   // the same network as SCL:
   MODE_MAINTENANCE_STATE_RESETTING:
   #tempDummy := FALSE;
END_REGION

REGION Network 68: Unit mode Maintenance - State Resetting
   RUNG wire#powerrail
      Contact( FALSE )
      S_Coil( "InstLPMLV2022_UnitModeStateManagerBool".SC )
   END_RUNG
   // the same network as SCL:
   IF FALSE THEN "InstLPMLV2022_UnitModeStateManagerBool".SC := TRUE; END_IF;
END_REGION

REGION Network 69: Unit mode Maintenance - State Resetting: Last network
   // Do not modify this network.
   RUNG wire#powerrail
      Contact( TRUE )
      JumpCoil( END )
   END_RUNG
   // the same network as SCL:
   IF TRUE THEN GOTO END; END_IF;
END_REGION

REGION Network 70: Unit mode Maintenance - State Idle: First network
   Label( MODE_MAINTENANCE_STATE_IDLE )
   RUNG wire#powerrail
      Contact( FALSE )
      Coil( #tempDummy )
   END_RUNG
   // the same network as SCL:
   MODE_MAINTENANCE_STATE_IDLE:
   #tempDummy := FALSE;
END_REGION

REGION Network 71: Unit mode Maintenance - State Idle
END_REGION

REGION Network 72: Unit mode Maintenance - State Idle: Last network
   // Do not modify this network.
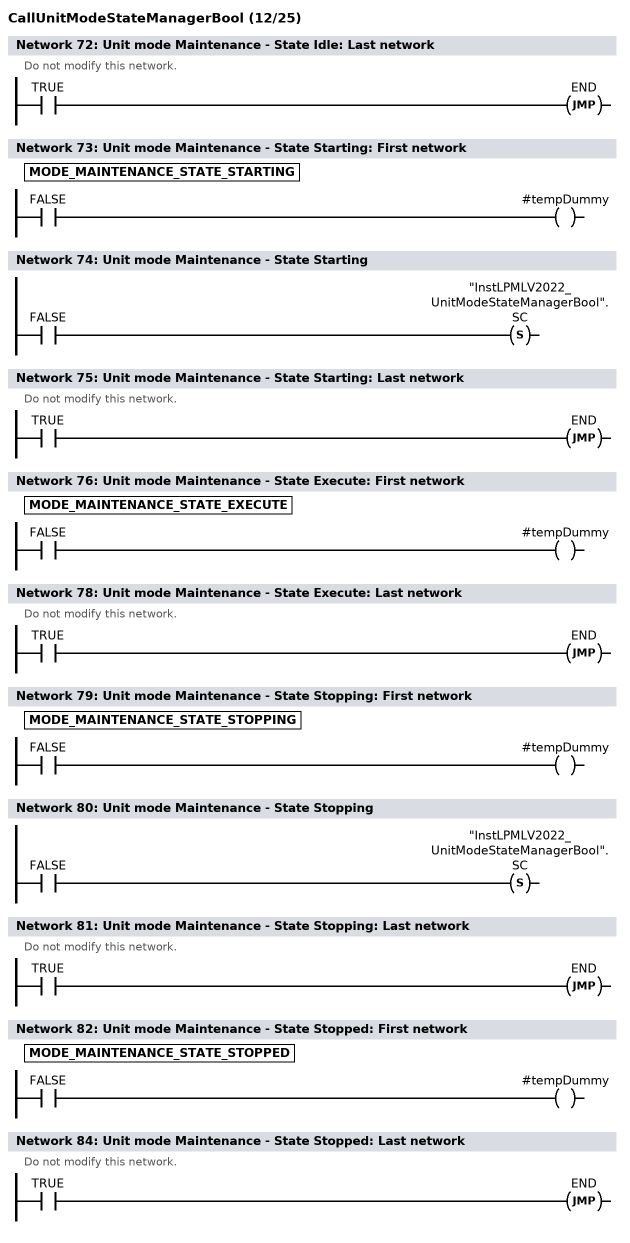
   RUNG wire#powerrail
      Contact( TRUE )
      JumpCoil( END )
   END_RUNG
   // the same network as SCL:
   IF TRUE THEN GOTO END; END_IF;
END_REGION

REGION Network 73: Unit mode Maintenance - State Starting: First network
   Label( MODE_MAINTENANCE_STATE_STARTING )
   RUNG wire#powerrail
      Contact( FALSE )
      Coil( #tempDummy )
   END_RUNG
   // the same network as SCL:
   MODE_MAINTENANCE_STATE_STARTING:
   #tempDummy := FALSE;
END_REGION

REGION Network 74: Unit mode Maintenance - State Starting
   RUNG wire#powerrail
      Contact( FALSE )
      S_Coil( "InstLPMLV2022_UnitModeStateManagerBool".SC )
   END_RUNG
   // the same network as SCL:
   IF FALSE THEN "InstLPMLV2022_UnitModeStateManagerBool".SC := TRUE; END_IF;
END_REGION

REGION Network 75: Unit mode Maintenance - State Starting: Last network
   // Do not modify this network.
   RUNG wire#powerrail
      Contact( TRUE )
      JumpCoil( END )
   END_RUNG
   // the same network as SCL:
   IF TRUE THEN GOTO END; END_IF;
END_REGION

REGION Network 76: Unit mode Maintenance - State Execute: First network
   Label( MODE_MAINTENANCE_STATE_EXECUTE )
   RUNG wire#powerrail
      Contact( FALSE )
      Coil( #tempDummy )
   END_RUNG
   // the same network as SCL:
   MODE_MAINTENANCE_STATE_EXECUTE:
   #tempDummy := FALSE;
END_REGION

REGION Network 77: Unit mode Maintenance - State Execute
END_REGION

REGION Network 78: Unit mode Maintenance - State Execute: Last network
   // Do not modify this network.
   RUNG wire#powerrail
      Contact( TRUE )
      JumpCoil( END )
   END_RUNG
   // the same network as SCL:
   IF TRUE THEN GOTO END; END_IF;
END_REGION

REGION Network 79: Unit mode Maintenance - State Stopping: First network
   Label( MODE_MAINTENANCE_STATE_STOPPING )
   RUNG wire#powerrail
      Contact( FALSE )
      Coil( #tempDummy )
   END_RUNG
   // the same network as SCL:
   MODE_MAINTENANCE_STATE_STOPPING:
   #tempDummy := FALSE;
END_REGION

REGION Network 80: Unit mode Maintenance - State Stopping
   RUNG wire#powerrail
      Contact( FALSE )
      S_Coil( "InstLPMLV2022_UnitModeStateManagerBool".SC )
   END_RUNG
   // the same network as SCL:
   IF FALSE THEN "InstLPMLV2022_UnitModeStateManagerBool".SC := TRUE; END_IF;
END_REGION

REGION Network 81: Unit mode Maintenance - State Stopping: Last network
   // Do not modify this network.
   RUNG wire#powerrail
      Contact( TRUE )
      JumpCoil( END )
   END_RUNG
   // the same network as SCL:
   IF TRUE THEN GOTO END; END_IF;
END_REGION

REGION Network 82: Unit mode Maintenance - State Stopped: First network
   Label( MODE_MAINTENANCE_STATE_STOPPED )
   RUNG wire#powerrail
      Contact( FALSE )
      Coil( #tempDummy )
   END_RUNG
   // the same network as SCL:
   MODE_MAINTENANCE_STATE_STOPPED:
   #tempDummy := FALSE;
END_REGION

REGION Network 83: Unit mode Maintenance - State Stopped
END_REGION

REGION Network 84: Unit mode Maintenance - State Stopped: Last network
   // Do not modify this network.
   RUNG wire#powerrail
      Contact( TRUE )
      JumpCoil( END )
   END_RUNG
   // the same network as SCL:
   IF TRUE THEN GOTO END; END_IF;
END_REGION

REGION Network 85: Unit mode Maintenance - State Holding: First network
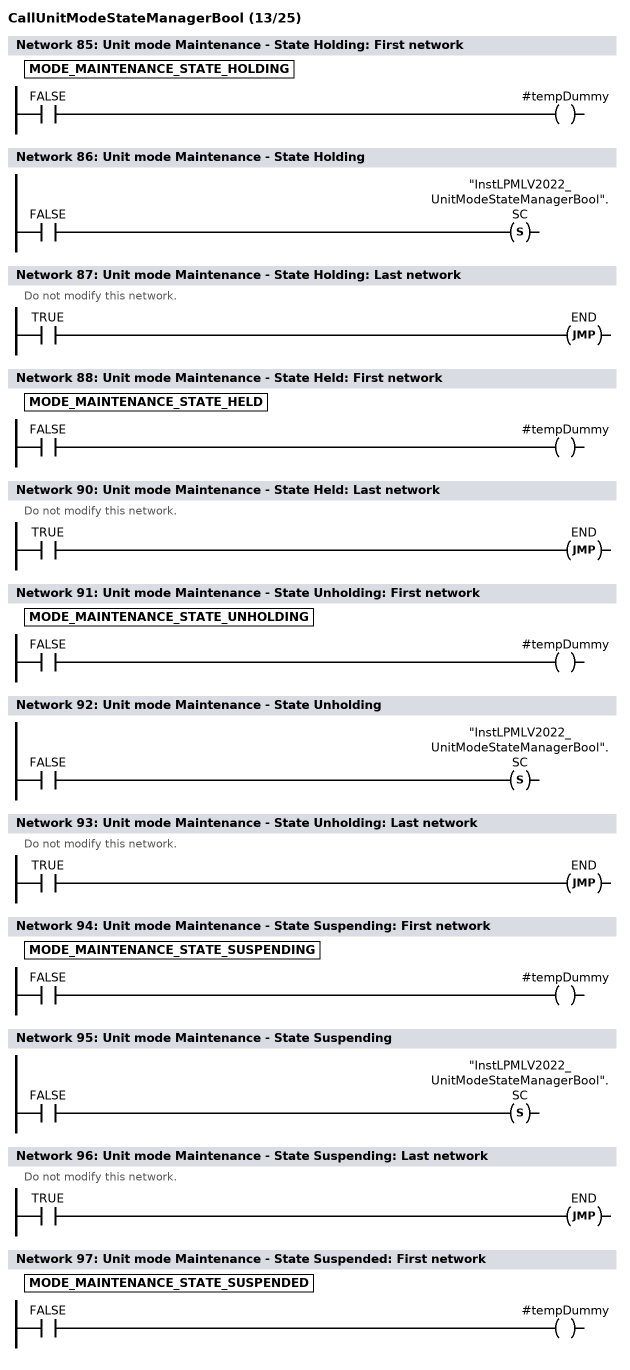
   Label( MODE_MAINTENANCE_STATE_HOLDING )
   RUNG wire#powerrail
      Contact( FALSE )
      Coil( #tempDummy )
   END_RUNG
   // the same network as SCL:
   MODE_MAINTENANCE_STATE_HOLDING:
   #tempDummy := FALSE;
END_REGION

REGION Network 86: Unit mode Maintenance - State Holding
   RUNG wire#powerrail
      Contact( FALSE )
      S_Coil( "InstLPMLV2022_UnitModeStateManagerBool".SC )
   END_RUNG
   // the same network as SCL:
   IF FALSE THEN "InstLPMLV2022_UnitModeStateManagerBool".SC := TRUE; END_IF;
END_REGION

REGION Network 87: Unit mode Maintenance - State Holding: Last network
   // Do not modify this network.
   RUNG wire#powerrail
      Contact( TRUE )
      JumpCoil( END )
   END_RUNG
   // the same network as SCL:
   IF TRUE THEN GOTO END; END_IF;
END_REGION

REGION Network 88: Unit mode Maintenance - State Held: First network
   Label( MODE_MAINTENANCE_STATE_HELD )
   RUNG wire#powerrail
      Contact( FALSE )
      Coil( #tempDummy )
   END_RUNG
   // the same network as SCL:
   MODE_MAINTENANCE_STATE_HELD:
   #tempDummy := FALSE;
END_REGION

REGION Network 89: Unit mode Maintenance - State Held
END_REGION

REGION Network 90: Unit mode Maintenance - State Held: Last network
   // Do not modify this network.
   RUNG wire#powerrail
      Contact( TRUE )
      JumpCoil( END )
   END_RUNG
   // the same network as SCL:
   IF TRUE THEN GOTO END; END_IF;
END_REGION

REGION Network 91: Unit mode Maintenance - State Unholding: First network
   Label( MODE_MAINTENANCE_STATE_UNHOLDING )
   RUNG wire#powerrail
      Contact( FALSE )
      Coil( #tempDummy )
   END_RUNG
   // the same network as SCL:
   MODE_MAINTENANCE_STATE_UNHOLDING:
   #tempDummy := FALSE;
END_REGION

REGION Network 92: Unit mode Maintenance - State Unholding
   RUNG wire#powerrail
      Contact( FALSE )
      S_Coil( "InstLPMLV2022_UnitModeStateManagerBool".SC )
   END_RUNG
   // the same network as SCL:
   IF FALSE THEN "InstLPMLV2022_UnitModeStateManagerBool".SC := TRUE; END_IF;
END_REGION

REGION Network 93: Unit mode Maintenance - State Unholding: Last network
   // Do not modify this network.
   RUNG wire#powerrail
      Contact( TRUE )
      JumpCoil( END )
   END_RUNG
   // the same network as SCL:
   IF TRUE THEN GOTO END; END_IF;
END_REGION

REGION Network 94: Unit mode Maintenance - State Suspending: First network
   Label( MODE_MAINTENANCE_STATE_SUSPENDING )
   RUNG wire#powerrail
      Contact( FALSE )
      Coil( #tempDummy )
   END_RUNG
   // the same network as SCL:
   MODE_MAINTENANCE_STATE_SUSPENDING:
   #tempDummy := FALSE;
END_REGION

REGION Network 95: Unit mode Maintenance - State Suspending
   RUNG wire#powerrail
      Contact( FALSE )
      S_Coil( "InstLPMLV2022_UnitModeStateManagerBool".SC )
   END_RUNG
   // the same network as SCL:
   IF FALSE THEN "InstLPMLV2022_UnitModeStateManagerBool".SC := TRUE; END_IF;
END_REGION

REGION Network 96: Unit mode Maintenance - State Suspending: Last network
   // Do not modify this network.
   RUNG wire#powerrail
      Contact( TRUE )
      JumpCoil( END )
   END_RUNG
   // the same network as SCL:
   IF TRUE THEN GOTO END; END_IF;
END_REGION

REGION Network 97: Unit mode Maintenance - State Suspended: First network
   Label( MODE_MAINTENANCE_STATE_SUSPENDED )
   RUNG wire#powerrail
      Contact( FALSE )
      Coil( #tempDummy )
   END_RUNG
   // the same network as SCL:
   MODE_MAINTENANCE_STATE_SUSPENDED:
   #tempDummy := FALSE;
END_REGION

REGION Network 98: Unit mode Maintenance - State Suspended
END_REGION

REGION Network 99: Unit mode Maintenance - State Suspended: Last network
   // Do not modify this network.
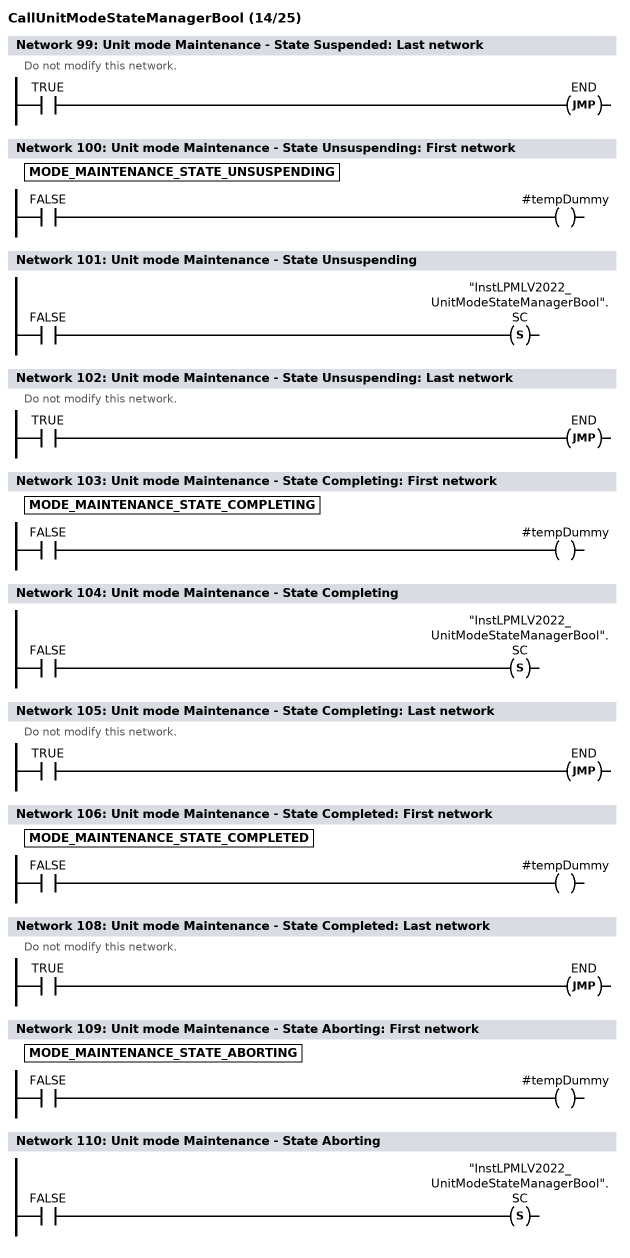
   RUNG wire#powerrail
      Contact( TRUE )
      JumpCoil( END )
   END_RUNG
   // the same network as SCL:
   IF TRUE THEN GOTO END; END_IF;
END_REGION

REGION Network 100: Unit mode Maintenance - State Unsuspending: First network
   Label( MODE_MAINTENANCE_STATE_UNSUSPENDING )
   RUNG wire#powerrail
      Contact( FALSE )
      Coil( #tempDummy )
   END_RUNG
   // the same network as SCL:
   MODE_MAINTENANCE_STATE_UNSUSPENDING:
   #tempDummy := FALSE;
END_REGION

REGION Network 101: Unit mode Maintenance - State Unsuspending
   RUNG wire#powerrail
      Contact( FALSE )
      S_Coil( "InstLPMLV2022_UnitModeStateManagerBool".SC )
   END_RUNG
   // the same network as SCL:
   IF FALSE THEN "InstLPMLV2022_UnitModeStateManagerBool".SC := TRUE; END_IF;
END_REGION

REGION Network 102: Unit mode Maintenance - State Unsuspending: Last network
   // Do not modify this network.
   RUNG wire#powerrail
      Contact( TRUE )
      JumpCoil( END )
   END_RUNG
   // the same network as SCL:
   IF TRUE THEN GOTO END; END_IF;
END_REGION

REGION Network 103: Unit mode Maintenance - State Completing: First network
   Label( MODE_MAINTENANCE_STATE_COMPLETING )
   RUNG wire#powerrail
      Contact( FALSE )
      Coil( #tempDummy )
   END_RUNG
   // the same network as SCL:
   MODE_MAINTENANCE_STATE_COMPLETING:
   #tempDummy := FALSE;
END_REGION

REGION Network 104: Unit mode Maintenance - State Completing
   RUNG wire#powerrail
      Contact( FALSE )
      S_Coil( "InstLPMLV2022_UnitModeStateManagerBool".SC )
   END_RUNG
   // the same network as SCL:
   IF FALSE THEN "InstLPMLV2022_UnitModeStateManagerBool".SC := TRUE; END_IF;
END_REGION

REGION Network 105: Unit mode Maintenance - State Completing: Last network
   // Do not modify this network.
   RUNG wire#powerrail
      Contact( TRUE )
      JumpCoil( END )
   END_RUNG
   // the same network as SCL:
   IF TRUE THEN GOTO END; END_IF;
END_REGION

REGION Network 106: Unit mode Maintenance - State Completed: First network
   Label( MODE_MAINTENANCE_STATE_COMPLETED )
   RUNG wire#powerrail
      Contact( FALSE )
      Coil( #tempDummy )
   END_RUNG
   // the same network as SCL:
   MODE_MAINTENANCE_STATE_COMPLETED:
   #tempDummy := FALSE;
END_REGION

REGION Network 107: Unit mode Maintenance - State Completed
END_REGION

REGION Network 108: Unit mode Maintenance - State Completed: Last network
   // Do not modify this network.
   RUNG wire#powerrail
      Contact( TRUE )
      JumpCoil( END )
   END_RUNG
   // the same network as SCL:
   IF TRUE THEN GOTO END; END_IF;
END_REGION

REGION Network 109: Unit mode Maintenance - State Aborting: First network
   Label( MODE_MAINTENANCE_STATE_ABORTING )
   RUNG wire#powerrail
      Contact( FALSE )
      Coil( #tempDummy )
   END_RUNG
   // the same network as SCL:
   MODE_MAINTENANCE_STATE_ABORTING:
   #tempDummy := FALSE;
END_REGION

REGION Network 110: Unit mode Maintenance - State Aborting
   RUNG wire#powerrail
      Contact( FALSE )
      S_Coil( "InstLPMLV2022_UnitModeStateManagerBool".SC )
   END_RUNG
   // the same network as SCL:
   IF FALSE THEN "InstLPMLV2022_UnitModeStateManagerBool".SC := TRUE; END_IF;
END_REGION

REGION Network 111: Unit mode Maintenance - State Aborting: Last network
   // Do not modify this network.
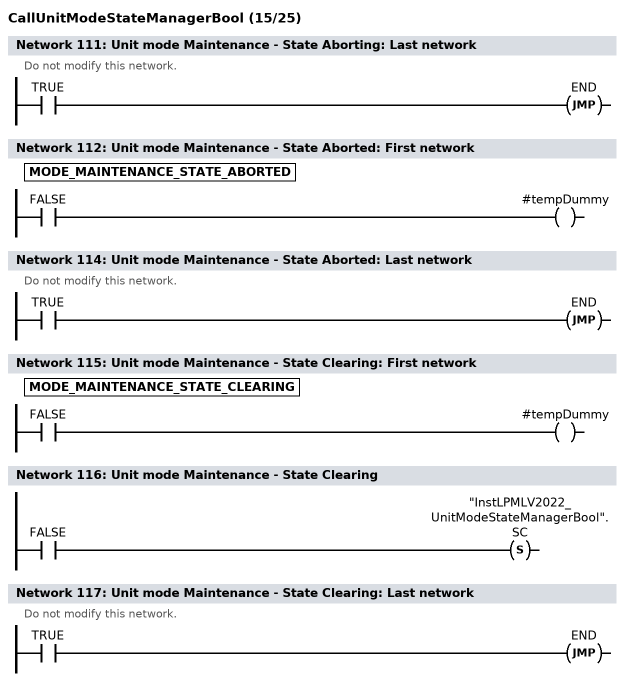
   RUNG wire#powerrail
      Contact( TRUE )
      JumpCoil( END )
   END_RUNG
   // the same network as SCL:
   IF TRUE THEN GOTO END; END_IF;
END_REGION

REGION Network 112: Unit mode Maintenance - State Aborted: First network
   Label( MODE_MAINTENANCE_STATE_ABORTED )
   RUNG wire#powerrail
      Contact( FALSE )
      Coil( #tempDummy )
   END_RUNG
   // the same network as SCL:
   MODE_MAINTENANCE_STATE_ABORTED:
   #tempDummy := FALSE;
END_REGION

REGION Network 113: Unit mode Maintenance - State Aborted
END_REGION

REGION Network 114: Unit mode Maintenance - State Aborted: Last network
   // Do not modify this network.
   RUNG wire#powerrail
      Contact( TRUE )
      JumpCoil( END )
   END_RUNG
   // the same network as SCL:
   IF TRUE THEN GOTO END; END_IF;
END_REGION

REGION Network 115: Unit mode Maintenance - State Clearing: First network
   Label( MODE_MAINTENANCE_STATE_CLEARING )
   RUNG wire#powerrail
      Contact( FALSE )
      Coil( #tempDummy )
   END_RUNG
   // the same network as SCL:
   MODE_MAINTENANCE_STATE_CLEARING:
   #tempDummy := FALSE;
END_REGION

REGION Network 116: Unit mode Maintenance - State Clearing
   RUNG wire#powerrail
      Contact( FALSE )
      S_Coil( "InstLPMLV2022_UnitModeStateManagerBool".SC )
   END_RUNG
   // the same network as SCL:
   IF FALSE THEN "InstLPMLV2022_UnitModeStateManagerBool".SC := TRUE; END_IF;
END_REGION

REGION Network 117: Unit mode Maintenance - State Clearing: Last network
   // Do not modify this network.
   RUNG wire#powerrail
      Contact( TRUE )
      JumpCoil( END )
   END_RUNG
   // the same network as SCL:
   IF TRUE THEN GOTO END; END_IF;
END_REGION

REGION Network 118: Unit mode Manual - Decode current state for unit mode (1/2)
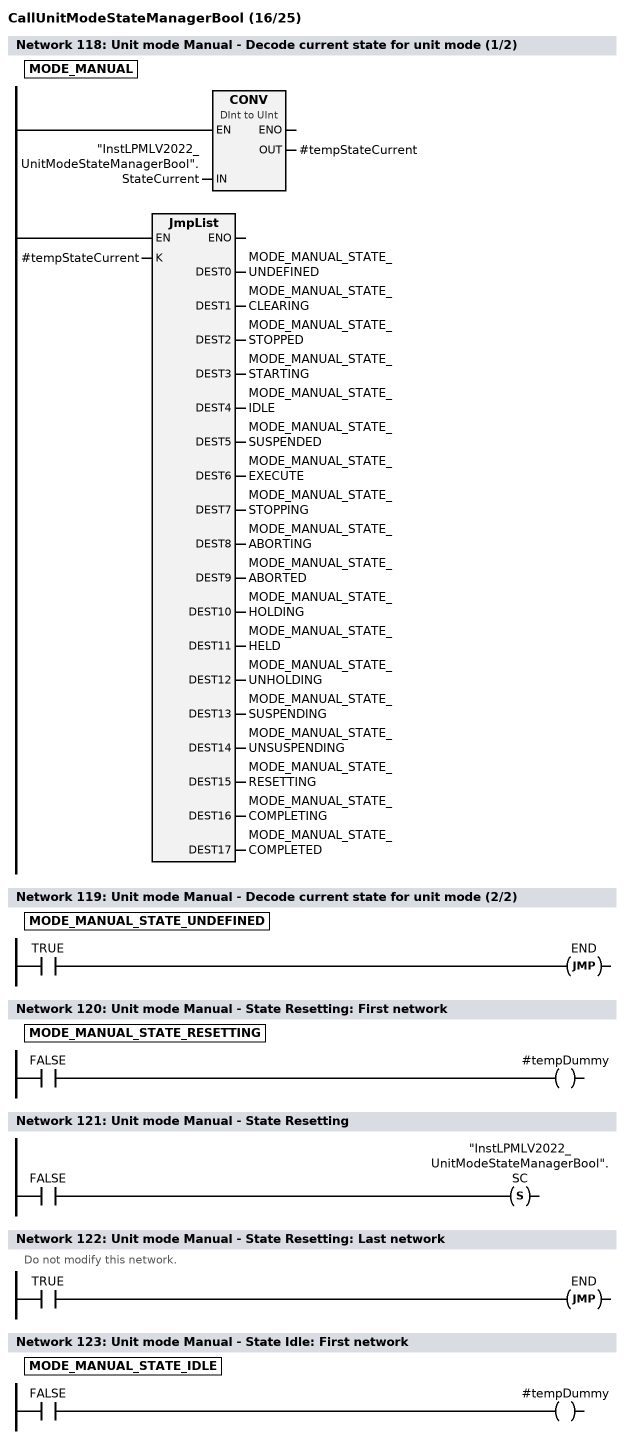
   // no SCL statement known for JmpList: written as a call
   MODE_MANUAL:
   #tempStateCurrent := DINT_TO_UINT("InstLPMLV2022_UnitModeStateManagerBool".StateCurrent);
   JmpList(k := #tempStateCurrent,
           dest0 => MODE_MANUAL_STATE_UNDEFINED,
           dest1 => MODE_MANUAL_STATE_CLEARING,
           dest2 => MODE_MANUAL_STATE_STOPPED,
           dest3 => MODE_MANUAL_STATE_STARTING,
           dest4 => MODE_MANUAL_STATE_IDLE,
           dest5 => MODE_MANUAL_STATE_SUSPENDED,
           dest6 => MODE_MANUAL_STATE_EXECUTE,
           dest7 => MODE_MANUAL_STATE_STOPPING,
           dest8 => MODE_MANUAL_STATE_ABORTING,
           dest9 => MODE_MANUAL_STATE_ABORTED,
           dest10 => MODE_MANUAL_STATE_HOLDING,
           dest11 => MODE_MANUAL_STATE_HELD,
           dest12 => MODE_MANUAL_STATE_UNHOLDING,
           dest13 => MODE_MANUAL_STATE_SUSPENDING,
           dest14 => MODE_MANUAL_STATE_UNSUSPENDING,
           dest15 => MODE_MANUAL_STATE_RESETTING,
           dest16 => MODE_MANUAL_STATE_COMPLETING,
           dest17 => MODE_MANUAL_STATE_COMPLETED);
END_REGION

REGION Network 119: Unit mode Manual - Decode current state for unit mode (2/2)
   Label( MODE_MANUAL_STATE_UNDEFINED )
   RUNG wire#powerrail
      Contact( TRUE )
      JumpCoil( END )
   END_RUNG
   // the same network as SCL:
   MODE_MANUAL_STATE_UNDEFINED:
   IF TRUE THEN GOTO END; END_IF;
END_REGION

REGION Network 120: Unit mode Manual - State Resetting: First network
   Label( MODE_MANUAL_STATE_RESETTING )
   RUNG wire#powerrail
      Contact( FALSE )
      Coil( #tempDummy )
   END_RUNG
   // the same network as SCL:
   MODE_MANUAL_STATE_RESETTING:
   #tempDummy := FALSE;
END_REGION

REGION Network 121: Unit mode Manual - State Resetting
   RUNG wire#powerrail
      Contact( FALSE )
      S_Coil( "InstLPMLV2022_UnitModeStateManagerBool".SC )
   END_RUNG
   // the same network as SCL:
   IF FALSE THEN "InstLPMLV2022_UnitModeStateManagerBool".SC := TRUE; END_IF;
END_REGION

REGION Network 122: Unit mode Manual - State Resetting: Last network
   // Do not modify this network.
   RUNG wire#powerrail
      Contact( TRUE )
      JumpCoil( END )
   END_RUNG
   // the same network as SCL:
   IF TRUE THEN GOTO END; END_IF;
END_REGION

REGION Network 123: Unit mode Manual - State Idle: First network
   Label( MODE_MANUAL_STATE_IDLE )
   RUNG wire#powerrail
      Contact( FALSE )
      Coil( #tempDummy )
   END_RUNG
   // the same network as SCL:
   MODE_MANUAL_STATE_IDLE:
   #tempDummy := FALSE;
END_REGION

REGION Network 124: Unit mode Manual - State Idle
END_REGION

REGION Network 125: Unit mode Manual - State Idle: Last network
   // Do not modify this network.
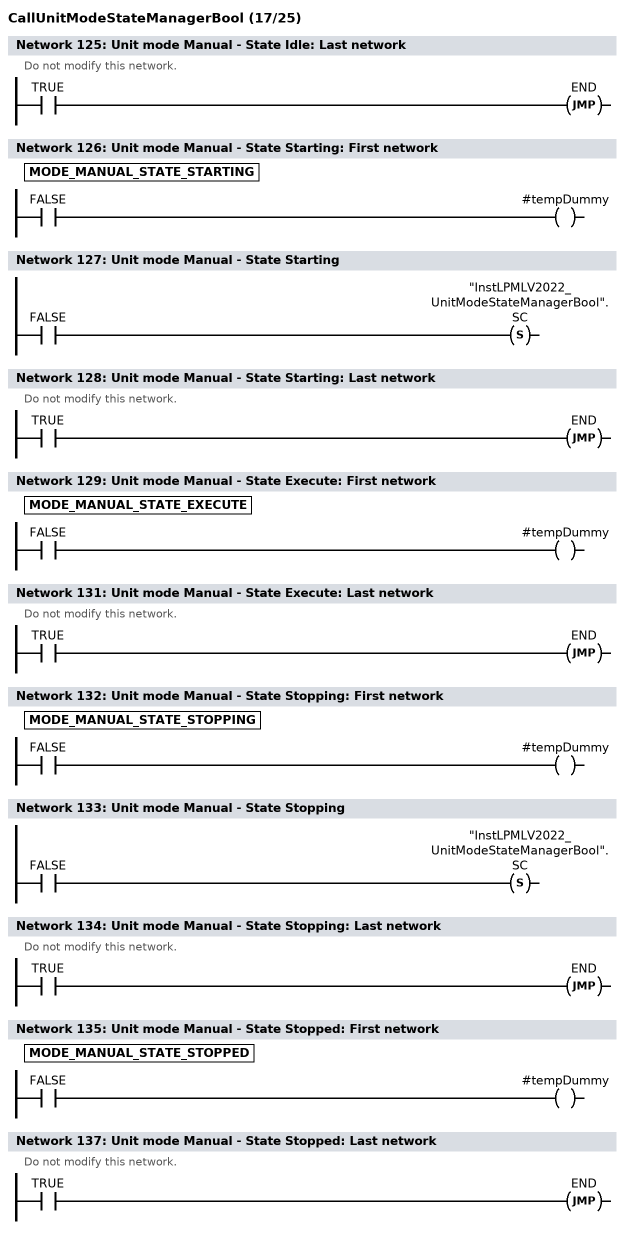
   RUNG wire#powerrail
      Contact( TRUE )
      JumpCoil( END )
   END_RUNG
   // the same network as SCL:
   IF TRUE THEN GOTO END; END_IF;
END_REGION

REGION Network 126: Unit mode Manual - State Starting: First network
   Label( MODE_MANUAL_STATE_STARTING )
   RUNG wire#powerrail
      Contact( FALSE )
      Coil( #tempDummy )
   END_RUNG
   // the same network as SCL:
   MODE_MANUAL_STATE_STARTING:
   #tempDummy := FALSE;
END_REGION

REGION Network 127: Unit mode Manual - State Starting
   RUNG wire#powerrail
      Contact( FALSE )
      S_Coil( "InstLPMLV2022_UnitModeStateManagerBool".SC )
   END_RUNG
   // the same network as SCL:
   IF FALSE THEN "InstLPMLV2022_UnitModeStateManagerBool".SC := TRUE; END_IF;
END_REGION

REGION Network 128: Unit mode Manual - State Starting: Last network
   // Do not modify this network.
   RUNG wire#powerrail
      Contact( TRUE )
      JumpCoil( END )
   END_RUNG
   // the same network as SCL:
   IF TRUE THEN GOTO END; END_IF;
END_REGION

REGION Network 129: Unit mode Manual - State Execute: First network
   Label( MODE_MANUAL_STATE_EXECUTE )
   RUNG wire#powerrail
      Contact( FALSE )
      Coil( #tempDummy )
   END_RUNG
   // the same network as SCL:
   MODE_MANUAL_STATE_EXECUTE:
   #tempDummy := FALSE;
END_REGION

REGION Network 130: Unit mode Manual - State Execute
END_REGION

REGION Network 131: Unit mode Manual - State Execute: Last network
   // Do not modify this network.
   RUNG wire#powerrail
      Contact( TRUE )
      JumpCoil( END )
   END_RUNG
   // the same network as SCL:
   IF TRUE THEN GOTO END; END_IF;
END_REGION

REGION Network 132: Unit mode Manual - State Stopping: First network
   Label( MODE_MANUAL_STATE_STOPPING )
   RUNG wire#powerrail
      Contact( FALSE )
      Coil( #tempDummy )
   END_RUNG
   // the same network as SCL:
   MODE_MANUAL_STATE_STOPPING:
   #tempDummy := FALSE;
END_REGION

REGION Network 133: Unit mode Manual - State Stopping
   RUNG wire#powerrail
      Contact( FALSE )
      S_Coil( "InstLPMLV2022_UnitModeStateManagerBool".SC )
   END_RUNG
   // the same network as SCL:
   IF FALSE THEN "InstLPMLV2022_UnitModeStateManagerBool".SC := TRUE; END_IF;
END_REGION

REGION Network 134: Unit mode Manual - State Stopping: Last network
   // Do not modify this network.
   RUNG wire#powerrail
      Contact( TRUE )
      JumpCoil( END )
   END_RUNG
   // the same network as SCL:
   IF TRUE THEN GOTO END; END_IF;
END_REGION

REGION Network 135: Unit mode Manual - State Stopped: First network
   Label( MODE_MANUAL_STATE_STOPPED )
   RUNG wire#powerrail
      Contact( FALSE )
      Coil( #tempDummy )
   END_RUNG
   // the same network as SCL:
   MODE_MANUAL_STATE_STOPPED:
   #tempDummy := FALSE;
END_REGION

REGION Network 136: Unit mode Manual - State Stopped
END_REGION

REGION Network 137: Unit mode Manual - State Stopped: Last network
   // Do not modify this network.
   RUNG wire#powerrail
      Contact( TRUE )
      JumpCoil( END )
   END_RUNG
   // the same network as SCL:
   IF TRUE THEN GOTO END; END_IF;
END_REGION

REGION Network 138: Unit mode Manual - State Holding: First network
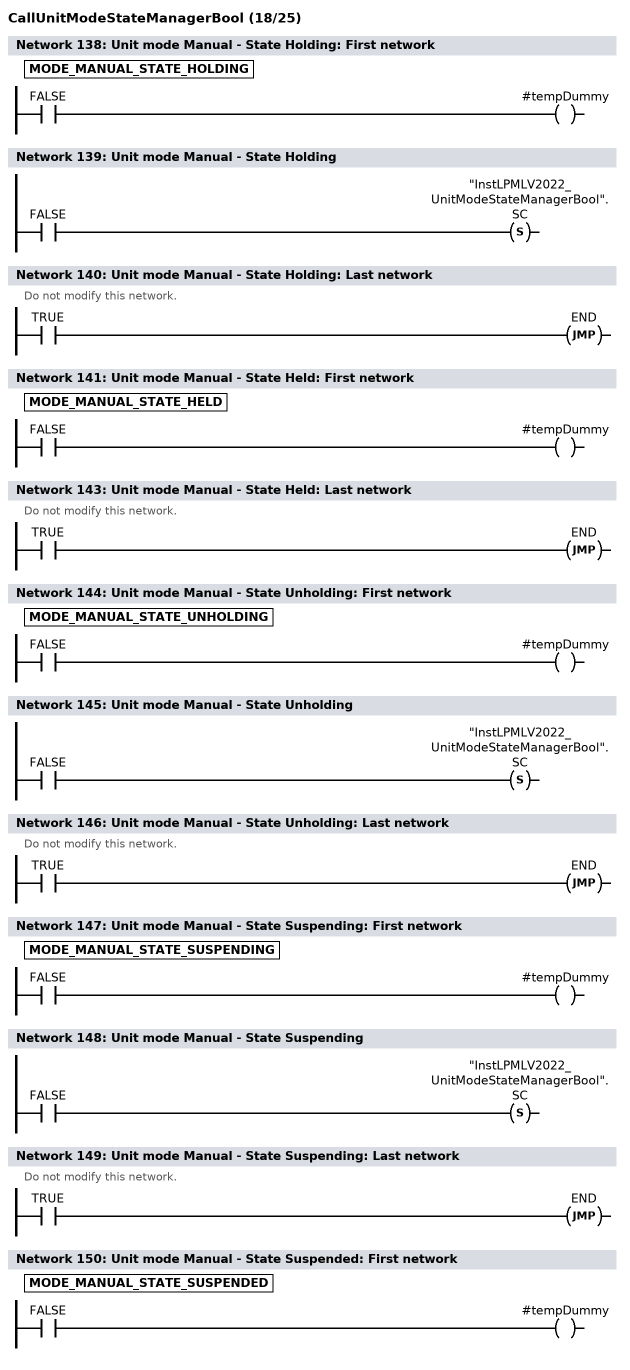
   Label( MODE_MANUAL_STATE_HOLDING )
   RUNG wire#powerrail
      Contact( FALSE )
      Coil( #tempDummy )
   END_RUNG
   // the same network as SCL:
   MODE_MANUAL_STATE_HOLDING:
   #tempDummy := FALSE;
END_REGION

REGION Network 139: Unit mode Manual - State Holding
   RUNG wire#powerrail
      Contact( FALSE )
      S_Coil( "InstLPMLV2022_UnitModeStateManagerBool".SC )
   END_RUNG
   // the same network as SCL:
   IF FALSE THEN "InstLPMLV2022_UnitModeStateManagerBool".SC := TRUE; END_IF;
END_REGION

REGION Network 140: Unit mode Manual - State Holding: Last network
   // Do not modify this network.
   RUNG wire#powerrail
      Contact( TRUE )
      JumpCoil( END )
   END_RUNG
   // the same network as SCL:
   IF TRUE THEN GOTO END; END_IF;
END_REGION

REGION Network 141: Unit mode Manual - State Held: First network
   Label( MODE_MANUAL_STATE_HELD )
   RUNG wire#powerrail
      Contact( FALSE )
      Coil( #tempDummy )
   END_RUNG
   // the same network as SCL:
   MODE_MANUAL_STATE_HELD:
   #tempDummy := FALSE;
END_REGION

REGION Network 142: Unit mode Manual - State Held
END_REGION

REGION Network 143: Unit mode Manual - State Held: Last network
   // Do not modify this network.
   RUNG wire#powerrail
      Contact( TRUE )
      JumpCoil( END )
   END_RUNG
   // the same network as SCL:
   IF TRUE THEN GOTO END; END_IF;
END_REGION

REGION Network 144: Unit mode Manual - State Unholding: First network
   Label( MODE_MANUAL_STATE_UNHOLDING )
   RUNG wire#powerrail
      Contact( FALSE )
      Coil( #tempDummy )
   END_RUNG
   // the same network as SCL:
   MODE_MANUAL_STATE_UNHOLDING:
   #tempDummy := FALSE;
END_REGION

REGION Network 145: Unit mode Manual - State Unholding
   RUNG wire#powerrail
      Contact( FALSE )
      S_Coil( "InstLPMLV2022_UnitModeStateManagerBool".SC )
   END_RUNG
   // the same network as SCL:
   IF FALSE THEN "InstLPMLV2022_UnitModeStateManagerBool".SC := TRUE; END_IF;
END_REGION

REGION Network 146: Unit mode Manual - State Unholding: Last network
   // Do not modify this network.
   RUNG wire#powerrail
      Contact( TRUE )
      JumpCoil( END )
   END_RUNG
   // the same network as SCL:
   IF TRUE THEN GOTO END; END_IF;
END_REGION

REGION Network 147: Unit mode Manual - State Suspending: First network
   Label( MODE_MANUAL_STATE_SUSPENDING )
   RUNG wire#powerrail
      Contact( FALSE )
      Coil( #tempDummy )
   END_RUNG
   // the same network as SCL:
   MODE_MANUAL_STATE_SUSPENDING:
   #tempDummy := FALSE;
END_REGION

REGION Network 148: Unit mode Manual - State Suspending
   RUNG wire#powerrail
      Contact( FALSE )
      S_Coil( "InstLPMLV2022_UnitModeStateManagerBool".SC )
   END_RUNG
   // the same network as SCL:
   IF FALSE THEN "InstLPMLV2022_UnitModeStateManagerBool".SC := TRUE; END_IF;
END_REGION

REGION Network 149: Unit mode Manual - State Suspending: Last network
   // Do not modify this network.
   RUNG wire#powerrail
      Contact( TRUE )
      JumpCoil( END )
   END_RUNG
   // the same network as SCL:
   IF TRUE THEN GOTO END; END_IF;
END_REGION

REGION Network 150: Unit mode Manual - State Suspended: First network
   Label( MODE_MANUAL_STATE_SUSPENDED )
   RUNG wire#powerrail
      Contact( FALSE )
      Coil( #tempDummy )
   END_RUNG
   // the same network as SCL:
   MODE_MANUAL_STATE_SUSPENDED:
   #tempDummy := FALSE;
END_REGION

REGION Network 151: Unit mode Manual - State Suspended
END_REGION

REGION Network 152: Unit mode Manual - State Suspended: Last network
   // Do not modify this network.
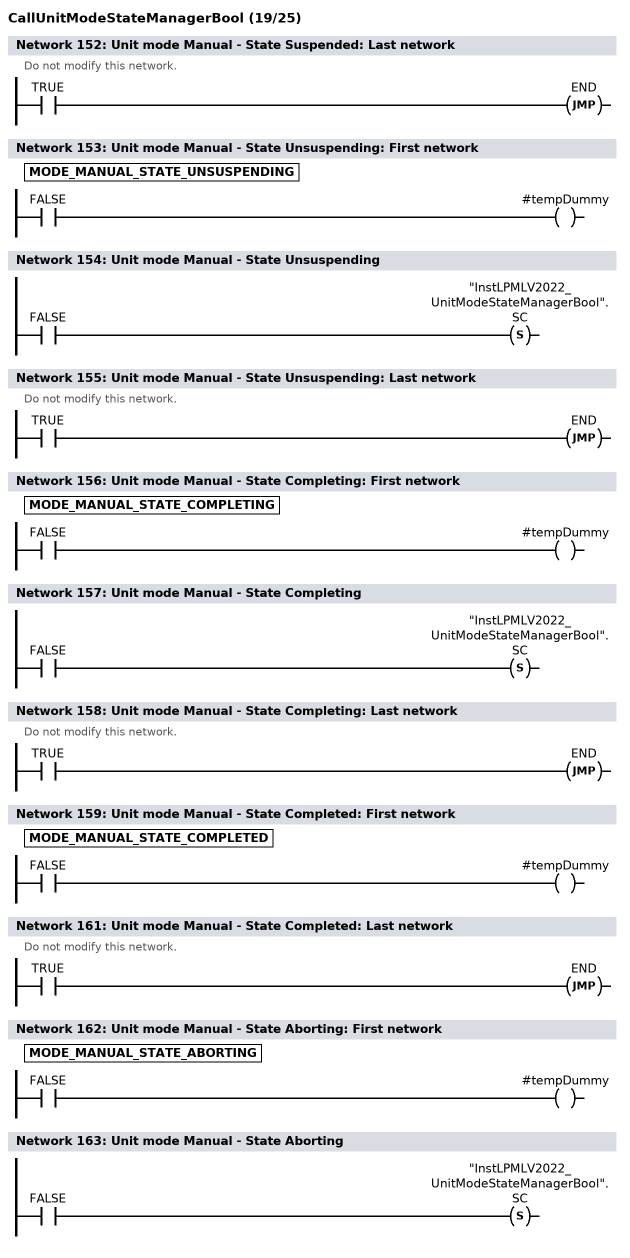
   RUNG wire#powerrail
      Contact( TRUE )
      JumpCoil( END )
   END_RUNG
   // the same network as SCL:
   IF TRUE THEN GOTO END; END_IF;
END_REGION

REGION Network 153: Unit mode Manual - State Unsuspending: First network
   Label( MODE_MANUAL_STATE_UNSUSPENDING )
   RUNG wire#powerrail
      Contact( FALSE )
      Coil( #tempDummy )
   END_RUNG
   // the same network as SCL:
   MODE_MANUAL_STATE_UNSUSPENDING:
   #tempDummy := FALSE;
END_REGION

REGION Network 154: Unit mode Manual - State Unsuspending
   RUNG wire#powerrail
      Contact( FALSE )
      S_Coil( "InstLPMLV2022_UnitModeStateManagerBool".SC )
   END_RUNG
   // the same network as SCL:
   IF FALSE THEN "InstLPMLV2022_UnitModeStateManagerBool".SC := TRUE; END_IF;
END_REGION

REGION Network 155: Unit mode Manual - State Unsuspending: Last network
   // Do not modify this network.
   RUNG wire#powerrail
      Contact( TRUE )
      JumpCoil( END )
   END_RUNG
   // the same network as SCL:
   IF TRUE THEN GOTO END; END_IF;
END_REGION

REGION Network 156: Unit mode Manual - State Completing: First network
   Label( MODE_MANUAL_STATE_COMPLETING )
   RUNG wire#powerrail
      Contact( FALSE )
      Coil( #tempDummy )
   END_RUNG
   // the same network as SCL:
   MODE_MANUAL_STATE_COMPLETING:
   #tempDummy := FALSE;
END_REGION

REGION Network 157: Unit mode Manual - State Completing
   RUNG wire#powerrail
      Contact( FALSE )
      S_Coil( "InstLPMLV2022_UnitModeStateManagerBool".SC )
   END_RUNG
   // the same network as SCL:
   IF FALSE THEN "InstLPMLV2022_UnitModeStateManagerBool".SC := TRUE; END_IF;
END_REGION

REGION Network 158: Unit mode Manual - State Completing: Last network
   // Do not modify this network.
   RUNG wire#powerrail
      Contact( TRUE )
      JumpCoil( END )
   END_RUNG
   // the same network as SCL:
   IF TRUE THEN GOTO END; END_IF;
END_REGION

REGION Network 159: Unit mode Manual - State Completed: First network
   Label( MODE_MANUAL_STATE_COMPLETED )
   RUNG wire#powerrail
      Contact( FALSE )
      Coil( #tempDummy )
   END_RUNG
   // the same network as SCL:
   MODE_MANUAL_STATE_COMPLETED:
   #tempDummy := FALSE;
END_REGION

REGION Network 160: Unit mode Manual - State Completed
END_REGION

REGION Network 161: Unit mode Manual - State Completed: Last network
   // Do not modify this network.
   RUNG wire#powerrail
      Contact( TRUE )
      JumpCoil( END )
   END_RUNG
   // the same network as SCL:
   IF TRUE THEN GOTO END; END_IF;
END_REGION

REGION Network 162: Unit mode Manual - State Aborting: First network
   Label( MODE_MANUAL_STATE_ABORTING )
   RUNG wire#powerrail
      Contact( FALSE )
      Coil( #tempDummy )
   END_RUNG
   // the same network as SCL:
   MODE_MANUAL_STATE_ABORTING:
   #tempDummy := FALSE;
END_REGION

REGION Network 163: Unit mode Manual - State Aborting
   RUNG wire#powerrail
      Contact( FALSE )
      S_Coil( "InstLPMLV2022_UnitModeStateManagerBool".SC )
   END_RUNG
   // the same network as SCL:
   IF FALSE THEN "InstLPMLV2022_UnitModeStateManagerBool".SC := TRUE; END_IF;
END_REGION

REGION Network 164: Unit mode Manual - State Aborting: Last network
   // Do not modify this network.
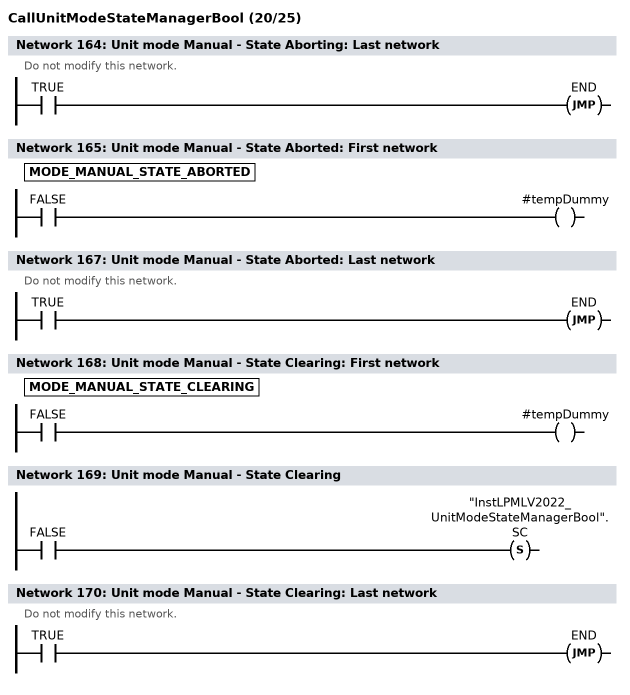
   RUNG wire#powerrail
      Contact( TRUE )
      JumpCoil( END )
   END_RUNG
   // the same network as SCL:
   IF TRUE THEN GOTO END; END_IF;
END_REGION

REGION Network 165: Unit mode Manual - State Aborted: First network
   Label( MODE_MANUAL_STATE_ABORTED )
   RUNG wire#powerrail
      Contact( FALSE )
      Coil( #tempDummy )
   END_RUNG
   // the same network as SCL:
   MODE_MANUAL_STATE_ABORTED:
   #tempDummy := FALSE;
END_REGION

REGION Network 166: Unit mode Manual - State Aborted
END_REGION

REGION Network 167: Unit mode Manual - State Aborted: Last network
   // Do not modify this network.
   RUNG wire#powerrail
      Contact( TRUE )
      JumpCoil( END )
   END_RUNG
   // the same network as SCL:
   IF TRUE THEN GOTO END; END_IF;
END_REGION

REGION Network 168: Unit mode Manual - State Clearing: First network
   Label( MODE_MANUAL_STATE_CLEARING )
   RUNG wire#powerrail
      Contact( FALSE )
      Coil( #tempDummy )
   END_RUNG
   // the same network as SCL:
   MODE_MANUAL_STATE_CLEARING:
   #tempDummy := FALSE;
END_REGION

REGION Network 169: Unit mode Manual - State Clearing
   RUNG wire#powerrail
      Contact( FALSE )
      S_Coil( "InstLPMLV2022_UnitModeStateManagerBool".SC )
   END_RUNG
   // the same network as SCL:
   IF FALSE THEN "InstLPMLV2022_UnitModeStateManagerBool".SC := TRUE; END_IF;
END_REGION

REGION Network 170: Unit mode Manual - State Clearing: Last network
   // Do not modify this network.
   RUNG wire#powerrail
      Contact( TRUE )
      JumpCoil( END )
   END_RUNG
   // the same network as SCL:
   IF TRUE THEN GOTO END; END_IF;
END_REGION

REGION Network 171: Unit mode User01 - Decode current state for unit mode (1/2)
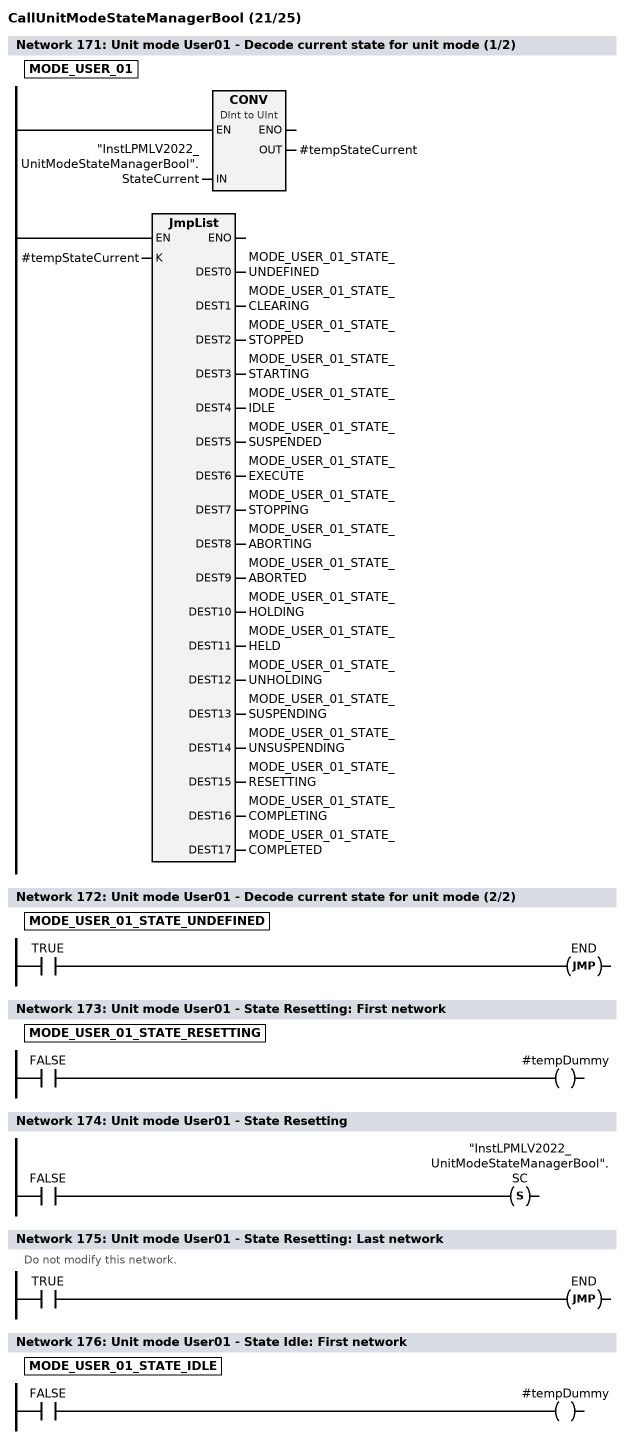
   // no SCL statement known for JmpList: written as a call
   MODE_USER_01:
   #tempStateCurrent := DINT_TO_UINT("InstLPMLV2022_UnitModeStateManagerBool".StateCurrent);
   JmpList(k := #tempStateCurrent,
           dest0 => MODE_USER_01_STATE_UNDEFINED,
           dest1 => MODE_USER_01_STATE_CLEARING,
           dest2 => MODE_USER_01_STATE_STOPPED,
           dest3 => MODE_USER_01_STATE_STARTING,
           dest4 => MODE_USER_01_STATE_IDLE,
           dest5 => MODE_USER_01_STATE_SUSPENDED,
           dest6 => MODE_USER_01_STATE_EXECUTE,
           dest7 => MODE_USER_01_STATE_STOPPING,
           dest8 => MODE_USER_01_STATE_ABORTING,
           dest9 => MODE_USER_01_STATE_ABORTED,
           dest10 => MODE_USER_01_STATE_HOLDING,
           dest11 => MODE_USER_01_STATE_HELD,
           dest12 => MODE_USER_01_STATE_UNHOLDING,
           dest13 => MODE_USER_01_STATE_SUSPENDING,
           dest14 => MODE_USER_01_STATE_UNSUSPENDING,
           dest15 => MODE_USER_01_STATE_RESETTING,
           dest16 => MODE_USER_01_STATE_COMPLETING,
           dest17 => MODE_USER_01_STATE_COMPLETED);
END_REGION

REGION Network 172: Unit mode User01 - Decode current state for unit mode (2/2)
   Label( MODE_USER_01_STATE_UNDEFINED )
   RUNG wire#powerrail
      Contact( TRUE )
      JumpCoil( END )
   END_RUNG
   // the same network as SCL:
   MODE_USER_01_STATE_UNDEFINED:
   IF TRUE THEN GOTO END; END_IF;
END_REGION

REGION Network 173: Unit mode User01 - State Resetting: First network
   Label( MODE_USER_01_STATE_RESETTING )
   RUNG wire#powerrail
      Contact( FALSE )
      Coil( #tempDummy )
   END_RUNG
   // the same network as SCL:
   MODE_USER_01_STATE_RESETTING:
   #tempDummy := FALSE;
END_REGION

REGION Network 174: Unit mode User01 - State Resetting
   RUNG wire#powerrail
      Contact( FALSE )
      S_Coil( "InstLPMLV2022_UnitModeStateManagerBool".SC )
   END_RUNG
   // the same network as SCL:
   IF FALSE THEN "InstLPMLV2022_UnitModeStateManagerBool".SC := TRUE; END_IF;
END_REGION

REGION Network 175: Unit mode User01 - State Resetting: Last network
   // Do not modify this network.
   RUNG wire#powerrail
      Contact( TRUE )
      JumpCoil( END )
   END_RUNG
   // the same network as SCL:
   IF TRUE THEN GOTO END; END_IF;
END_REGION

REGION Network 176: Unit mode User01 - State Idle: First network
   Label( MODE_USER_01_STATE_IDLE )
   RUNG wire#powerrail
      Contact( FALSE )
      Coil( #tempDummy )
   END_RUNG
   // the same network as SCL:
   MODE_USER_01_STATE_IDLE:
   #tempDummy := FALSE;
END_REGION

REGION Network 177: Unit mode User01 - State Idle
END_REGION

REGION Network 178: Unit mode User01 - State Idle: Last network
   // Do not modify this network.
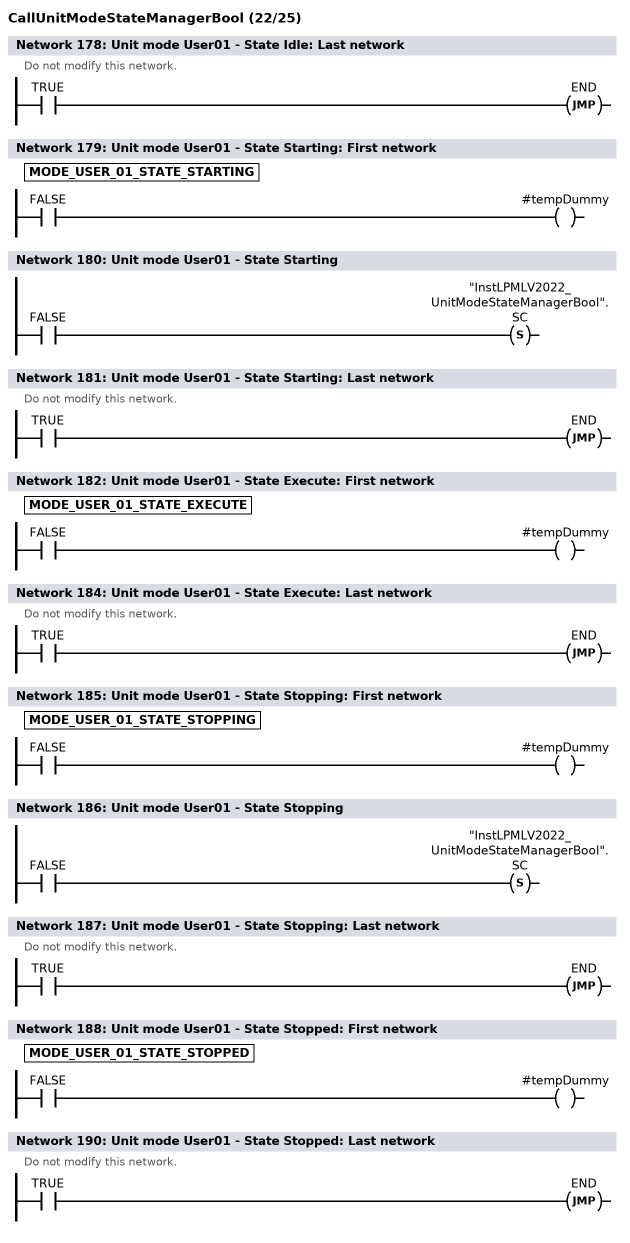
   RUNG wire#powerrail
      Contact( TRUE )
      JumpCoil( END )
   END_RUNG
   // the same network as SCL:
   IF TRUE THEN GOTO END; END_IF;
END_REGION

REGION Network 179: Unit mode User01 - State Starting: First network
   Label( MODE_USER_01_STATE_STARTING )
   RUNG wire#powerrail
      Contact( FALSE )
      Coil( #tempDummy )
   END_RUNG
   // the same network as SCL:
   MODE_USER_01_STATE_STARTING:
   #tempDummy := FALSE;
END_REGION

REGION Network 180: Unit mode User01 - State Starting
   RUNG wire#powerrail
      Contact( FALSE )
      S_Coil( "InstLPMLV2022_UnitModeStateManagerBool".SC )
   END_RUNG
   // the same network as SCL:
   IF FALSE THEN "InstLPMLV2022_UnitModeStateManagerBool".SC := TRUE; END_IF;
END_REGION

REGION Network 181: Unit mode User01 - State Starting: Last network
   // Do not modify this network.
   RUNG wire#powerrail
      Contact( TRUE )
      JumpCoil( END )
   END_RUNG
   // the same network as SCL:
   IF TRUE THEN GOTO END; END_IF;
END_REGION

REGION Network 182: Unit mode User01 - State Execute: First network
   Label( MODE_USER_01_STATE_EXECUTE )
   RUNG wire#powerrail
      Contact( FALSE )
      Coil( #tempDummy )
   END_RUNG
   // the same network as SCL:
   MODE_USER_01_STATE_EXECUTE:
   #tempDummy := FALSE;
END_REGION

REGION Network 183: Unit mode User01 - State Execute
END_REGION

REGION Network 184: Unit mode User01 - State Execute: Last network
   // Do not modify this network.
   RUNG wire#powerrail
      Contact( TRUE )
      JumpCoil( END )
   END_RUNG
   // the same network as SCL:
   IF TRUE THEN GOTO END; END_IF;
END_REGION

REGION Network 185: Unit mode User01 - State Stopping: First network
   Label( MODE_USER_01_STATE_STOPPING )
   RUNG wire#powerrail
      Contact( FALSE )
      Coil( #tempDummy )
   END_RUNG
   // the same network as SCL:
   MODE_USER_01_STATE_STOPPING:
   #tempDummy := FALSE;
END_REGION

REGION Network 186: Unit mode User01 - State Stopping
   RUNG wire#powerrail
      Contact( FALSE )
      S_Coil( "InstLPMLV2022_UnitModeStateManagerBool".SC )
   END_RUNG
   // the same network as SCL:
   IF FALSE THEN "InstLPMLV2022_UnitModeStateManagerBool".SC := TRUE; END_IF;
END_REGION

REGION Network 187: Unit mode User01 - State Stopping: Last network
   // Do not modify this network.
   RUNG wire#powerrail
      Contact( TRUE )
      JumpCoil( END )
   END_RUNG
   // the same network as SCL:
   IF TRUE THEN GOTO END; END_IF;
END_REGION

REGION Network 188: Unit mode User01 - State Stopped: First network
   Label( MODE_USER_01_STATE_STOPPED )
   RUNG wire#powerrail
      Contact( FALSE )
      Coil( #tempDummy )
   END_RUNG
   // the same network as SCL:
   MODE_USER_01_STATE_STOPPED:
   #tempDummy := FALSE;
END_REGION

REGION Network 189: Unit mode User01 - State Stopped
END_REGION

REGION Network 190: Unit mode User01 - State Stopped: Last network
   // Do not modify this network.
   RUNG wire#powerrail
      Contact( TRUE )
      JumpCoil( END )
   END_RUNG
   // the same network as SCL:
   IF TRUE THEN GOTO END; END_IF;
END_REGION

REGION Network 191: Unit mode User01 - State Holding: First network
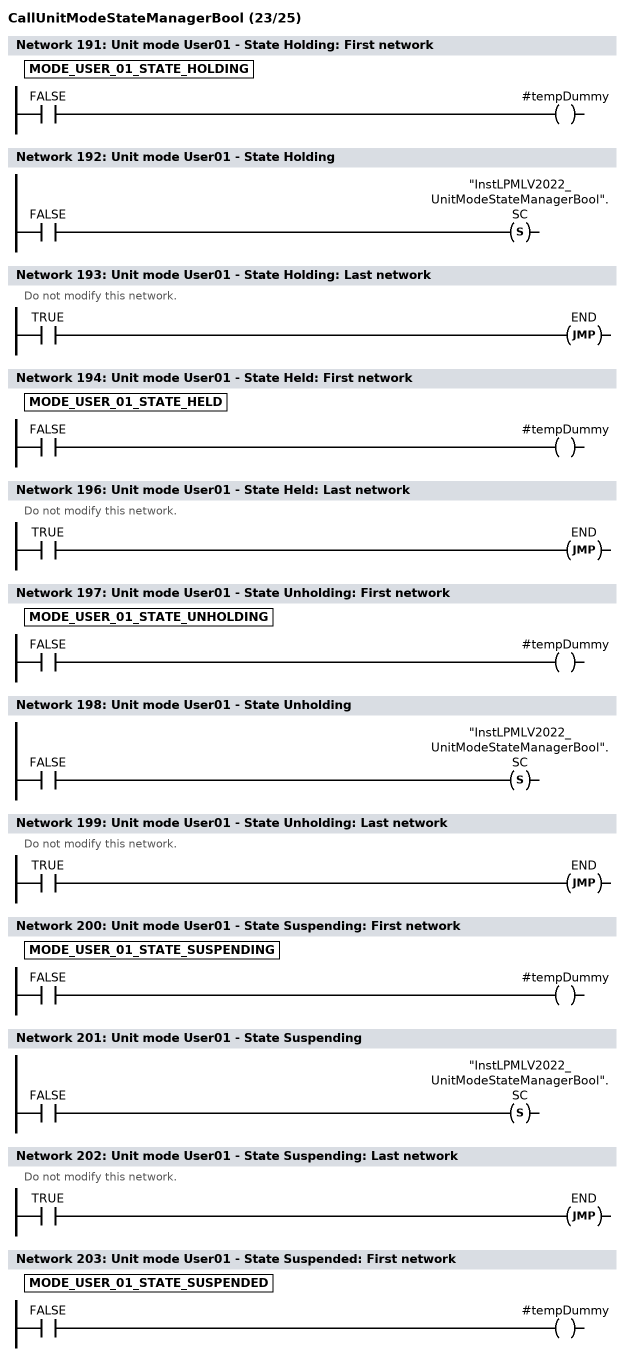
   Label( MODE_USER_01_STATE_HOLDING )
   RUNG wire#powerrail
      Contact( FALSE )
      Coil( #tempDummy )
   END_RUNG
   // the same network as SCL:
   MODE_USER_01_STATE_HOLDING:
   #tempDummy := FALSE;
END_REGION

REGION Network 192: Unit mode User01 - State Holding
   RUNG wire#powerrail
      Contact( FALSE )
      S_Coil( "InstLPMLV2022_UnitModeStateManagerBool".SC )
   END_RUNG
   // the same network as SCL:
   IF FALSE THEN "InstLPMLV2022_UnitModeStateManagerBool".SC := TRUE; END_IF;
END_REGION

REGION Network 193: Unit mode User01 - State Holding: Last network
   // Do not modify this network.
   RUNG wire#powerrail
      Contact( TRUE )
      JumpCoil( END )
   END_RUNG
   // the same network as SCL:
   IF TRUE THEN GOTO END; END_IF;
END_REGION

REGION Network 194: Unit mode User01 - State Held: First network
   Label( MODE_USER_01_STATE_HELD )
   RUNG wire#powerrail
      Contact( FALSE )
      Coil( #tempDummy )
   END_RUNG
   // the same network as SCL:
   MODE_USER_01_STATE_HELD:
   #tempDummy := FALSE;
END_REGION

REGION Network 195: Unit mode User01 - State Held
END_REGION

REGION Network 196: Unit mode User01 - State Held: Last network
   // Do not modify this network.
   RUNG wire#powerrail
      Contact( TRUE )
      JumpCoil( END )
   END_RUNG
   // the same network as SCL:
   IF TRUE THEN GOTO END; END_IF;
END_REGION

REGION Network 197: Unit mode User01 - State Unholding: First network
   Label( MODE_USER_01_STATE_UNHOLDING )
   RUNG wire#powerrail
      Contact( FALSE )
      Coil( #tempDummy )
   END_RUNG
   // the same network as SCL:
   MODE_USER_01_STATE_UNHOLDING:
   #tempDummy := FALSE;
END_REGION

REGION Network 198: Unit mode User01 - State Unholding
   RUNG wire#powerrail
      Contact( FALSE )
      S_Coil( "InstLPMLV2022_UnitModeStateManagerBool".SC )
   END_RUNG
   // the same network as SCL:
   IF FALSE THEN "InstLPMLV2022_UnitModeStateManagerBool".SC := TRUE; END_IF;
END_REGION

REGION Network 199: Unit mode User01 - State Unholding: Last network
   // Do not modify this network.
   RUNG wire#powerrail
      Contact( TRUE )
      JumpCoil( END )
   END_RUNG
   // the same network as SCL:
   IF TRUE THEN GOTO END; END_IF;
END_REGION

REGION Network 200: Unit mode User01 - State Suspending: First network
   Label( MODE_USER_01_STATE_SUSPENDING )
   RUNG wire#powerrail
      Contact( FALSE )
      Coil( #tempDummy )
   END_RUNG
   // the same network as SCL:
   MODE_USER_01_STATE_SUSPENDING:
   #tempDummy := FALSE;
END_REGION

REGION Network 201: Unit mode User01 - State Suspending
   RUNG wire#powerrail
      Contact( FALSE )
      S_Coil( "InstLPMLV2022_UnitModeStateManagerBool".SC )
   END_RUNG
   // the same network as SCL:
   IF FALSE THEN "InstLPMLV2022_UnitModeStateManagerBool".SC := TRUE; END_IF;
END_REGION

REGION Network 202: Unit mode User01 - State Suspending: Last network
   // Do not modify this network.
   RUNG wire#powerrail
      Contact( TRUE )
      JumpCoil( END )
   END_RUNG
   // the same network as SCL:
   IF TRUE THEN GOTO END; END_IF;
END_REGION

REGION Network 203: Unit mode User01 - State Suspended: First network
   Label( MODE_USER_01_STATE_SUSPENDED )
   RUNG wire#powerrail
      Contact( FALSE )
      Coil( #tempDummy )
   END_RUNG
   // the same network as SCL:
   MODE_USER_01_STATE_SUSPENDED:
   #tempDummy := FALSE;
END_REGION

REGION Network 204: Unit mode User01 - State Suspended
END_REGION

REGION Network 205: Unit mode User01 - State Suspended: Last network
   // Do not modify this network.
